C07301=1233.977,-39.079,-38.735,-179.809,5.259,148.853
C07302=1233.971,-38.829,-38.748,-179.806,5.259,148.852
C07303=1233.967,-38.579,-38.761,-179.804,5.260,148.851
C07304=1233.962,-38.330,-38.774,-179.802,5.259,148.851
C07305=1233.956,-38.080,-38.787,-179.799,5.260,148.850
C07306=1233.952,-37.831,-38.800,-179.797,5.260,148.849
C07307=1233.946,-37.581,-38.813,-179.794,5.260,148.849
C07308=1233.941,-37.331,-38.827,-179.792,5.261,148.848
C07309=1233.936,-37.082,-38.839,-179.789,5.260,148.847
C07310=1233.931,-36.832,-38.852,-179.787,5.261,148.846
C07311=1233.926,-36.582,-38.865,-179.785,5.261,148.846
C07312=1233.921,-36.333,-38.879,-179.782,5.261,148.845
C07313=1233.916,-36.083,-38.892,-179.779,5.262,148.844
C07314=1233.910,-35.834,-38.905,-179.777,5.261,148.844
C07315=1233.905,-35.584,-38.917,-179.775,5.262,148.843
C07316=1233.900,-35.334,-38.931,-179.773,5.261,148.842
C07317=1233.895,-35.085,-38.944,-179.769,5.262,148.841
C07318=1233.891,-34.835,-38.957,-179.767,5.262,148.841
C07319=1233.885,-34.586,-38.971,-179.765,5.262,148.840
C07320=1233.880,-34.336,-38.983,-179.762,5.262,148.839
C07321=1233.875,-34.086,-38.997,-179.760,5.262,148.839
C07322=1233.870,-33.837,-39.010,-179.757,5.262,148.838
C07323=1233.865,-33.587,-39.023,-179.755,5.263,148.837
C07324=1233.859,-33.338,-39.036,-179.753,5.263,148.836
C07325=1233.855,-33.088,-39.049,-179.750,5.263,148.836
C07326=1233.849,-32.839,-39.063,-179.748,5.263,148.835
C07327=1233.845,-32.589,-39.076,-179.745,5.263,148.834
C07328=1233.839,-32.339,-39.089,-179.742,5.264,148.834
C07329=1233.835,-32.090,-39.103,-179.740,5.263,148.833
C07330=1233.829,-31.840,-39.116,-179.738,5.264,148.832
C07331=1233.824,-31.590,-39.129,-179.736,5.264,148.832
C07332=1233.819,-31.341,-39.142,-179.733,5.264,148.831
C07333=1233.814,-31.092,-39.156,-179.730,5.265,148.830
C07334=1233.809,-30.842,-39.169,-179.728,5.264,148.829
C07335=1233.803,-30.593,-39.182,-179.725,5.265,148.829
C07336=1233.799,-30.343,-39.195,-179.723,5.264,148.828
C07337=1233.793,-30.093,-39.209,-179.720,5.265,148.827
C07338=1233.789,-29.844,-39.222,-179.718,5.265,148.826
C07339=1233.783,-29.594,-39.235,-179.716,5.265,148.826
C07340=1233.779,-29.344,-39.248,-179.713,5.265,148.825
C07341=1233.773,-29.095,-39.262,-179.711,5.265,148.824
C07342=1233.768,-28.845,-39.275,-179.708,5.266,148.824
C07343=1233.763,-28.596,-39.289,-179.705,5.266,148.823
C07344=1233.758,-28.346,-39.302,-179.703,5.266,148.822
C07345=1233.753,-28.096,-39.316,-179.701,5.266,148.822
C07346=1233.748,-27.846,-39.330,-179.698,5.267,148.821
C07347=1233.743,-27.596,-39.343,-179.696,5.267,148.820
C07348=1233.737,-27.347,-39.357,-179.693,5.267,148.819
C07349=1233.733,-27.097,-39.370,-179.691,5.267,148.819
C07350=1233.727,-26.848,-39.383,-179.689,5.267,148.818
C07351=1233.723,-26.598,-39.396,-179.686,5.268,148.817
C07352=1233.717,-26.349,-39.410,-179.683,5.267,148.816
C07353=1233.713,-26.099,-39.423,-179.681,5.268,148.816
C07354=1233.707,-25.850,-39.437,-179.679,5.267,148.815
C07355=1233.702,-25.600,-39.451,-179.676,5.268,148.814
C07356=1233.698,-25.351,-39.464,-179.673,5.268,148.814
C07357=1233.692,-25.101,-39.478,-179.671,5.268,148.813
C07358=1233.688,-24.852,-39.491,-179.669,5.269,148.812
C07359=1233.682,-24.602,-39.505,-179.666,5.269,148.812
C07360=1233.677,-24.352,-39.519,-179.664,5.269,148.811
C07361=1233.672,-24.103,-39.531,-179.661,5.269,148.810
C07362=1233.667,-23.853,-39.546,-179.659,5.269,148.809
C07363=1233.662,-23.603,-39.559,-179.656,5.269,148.809
C07364=1233.657,-23.354,-39.573,-179.654,5.270,148.808
C07365=1233.652,-23.104,-39.587,-179.652,5.270,148.807
C07366=1233.647,-22.855,-39.599,-179.649,5.270,148.807
C07367=1233.641,-22.586,-39.614,-179.646,5.270,148.806
C07368=1233.636,-22.316,-39.629,-179.643,5.271,148.805
C07369=1233.630,-22.047,-39.644,-179.641,5.271,148.804
C07370=1233.624,-21.778,-39.659,-179.638,5.271,148.804
C07371=1233.620,-21.528,-39.672,-179.635,5.271,148.803
C07372=1233.615,-21.278,-39.686,-179.633,5.271,148.802
C07373=1233.609,-21.029,-39.700,-179.631,5.271,148.801
C07374=1233.605,-20.779,-39.713,-179.628,5.272,148.801
C07375=1233.599,-20.530,-39.727,-179.626,5.272,148.800
C07376=1233.594,-20.281,-39.741,-179.623,5.272,148.799
C07377=1233.590,-20.031,-39.754,-179.620,5.273,148.799
C07378=1233.584,-19.782,-39.768,-179.618,5.272,148.798
C07379=1233.579,-19.532,-39.782,-179.616,5.273,148.797
C07380=1233.574,-19.282,-39.796,-179.614,5.273,148.796
C07381=1233.569,-19.033,-39.809,-179.611,5.273,148.796
C07382=1233.564,-18.783,-39.824,-179.608,5.274,148.795
C07383=1233.559,-18.533,-39.837,-179.606,5.273,148.794
C07384=1233.553,-18.284,-39.851,-179.604,5.274,148.794
C07385=1233.549,-18.035,-39.865,-179.601,5.274,148.793
C07386=1233.544,-17.784,-39.878,-179.599,5.274,148.792
C07387=1233.538,-17.535,-39.892,-179.596,5.275,148.792
C07388=1233.533,-17.285,-39.907,-179.594,5.275,148.791
C07389=1233.529,-17.036,-39.920,-179.591,5.275,148.790
C07390=1233.523,-16.786,-39.933,-179.589,5.275,148.790
C07391=1233.518,-16.537,-39.948,-179.586,5.275,148.789
C07392=1233.513,-16.287,-39.962,-179.584,5.275,148.788
C07393=1233.508,-16.038,-39.976,-179.581,5.276,148.787
C07394=1233.504,-15.789,-39.990,-179.579,5.275,148.787
C07395=1233.498,-15.538,-40.003,-179.576,5.276,148.786
C07396=1233.493,-15.289,-40.017,-179.574,5.276,148.785
C07397=1233.488,-15.040,-40.031,-179.571,5.276,148.784
C07398=1233.483,-14.790,-40.046,-179.569,5.277,148.784
C07399=1233.479,-14.540,-40.059,-179.566,5.277,148.783
C07400=1233.473,-14.291,-40.072,-179.564,5.277,148.782
C07401=1233.468,-14.041,-40.087,-179.561,5.277,148.782
C07402=1233.463,-13.791,-40.101,-179.559,5.278,148.781
C07403=1233.457,-13.542,-40.115,-179.557,5.278,148.780
C07404=1233.452,-13.293,-40.129,-179.554,5.278,148.780
C07405=1233.448,-13.043,-40.143,-179.551,5.279,148.779
C07406=1233.443,-12.794,-40.157,-179.549,5.278,148.778
C07407=1233.438,-12.545,-40.171,-179.547,5.279,148.777
C07408=1233.432,-12.294,-40.185,-179.544,5.279,148.777
C07409=1233.427,-12.045,-40.199,-179.542,5.279,148.776
C07410=1233.422,-11.795,-40.213,-179.539,5.280,148.775
C07411=1233.417,-11.546,-40.227,-179.537,5.280,148.775
C07412=1233.412,-11.296,-40.241,-179.534,5.279,148.774
C07413=1233.408,-11.047,-40.255,-179.531,5.280,148.773
C07414=1233.403,-10.797,-40.269,-179.529,5.280,148.772
C07415=1233.397,-10.548,-40.283,-179.527,5.280,148.772
C07416=1233.392,-10.298,-40.298,-179.524,5.281,148.771
C07417=1233.387,-10.049,-40.312,-179.521,5.281,148.770
C07418=1233.382,-9.799,-40.326,-179.519,5.281,148.770
C07419=1233.377,-9.550,-40.340,-179.517,5.281,148.769
C07420=1233.372,-9.300,-40.354,-179.514,5.282,148.768
C07421=1233.367,-9.050,-40.369,-179.512,5.282,148.768
C07422=1233.362,-8.801,-40.383,-179.509,5.282,148.767
C07423=1233.357,-8.551,-40.397,-179.506,5.283,148.766
C07424=1233.351,-8.302,-40.411,-179.504,5.282,148.765
C07425=1233.346,-8.052,-40.425,-179.502,5.283,148.765
C07426=1233.342,-7.803,-40.440,-179.499,5.283,148.764
C07427=1233.337,-7.553,-40.454,-179.497,5.283,148.763
C07428=1233.332,-7.303,-40.468,-179.494,5.284,148.763
C07429=1233.327,-7.053,-40.482,-179.492,5.284,148.762
C07430=1233.322,-6.805,-40.496,-179.490,5.284,148.761
C07431=1233.317,-6.555,-40.510,-179.487,5.284,148.761
C07432=1233.312,-6.305,-40.524,-179.484,5.285,148.760
C07433=1233.307,-6.056,-40.539,-179.482,5.286,148.759
C07434=1233.302,-5.806,-40.553,-179.480,5.285,148.759
C07435=1233.297,-5.556,-40.567,-179.477,5.286,148.758
C07436=1233.291,-5.307,-40.582,-179.474,5.286,148.757
C07437=1233.286,-5.058,-40.597,-179.472,5.286,148.756
C07438=1233.281,-4.808,-40.611,-179.469,5.286,148.756
C07439=1233.276,-4.558,-40.625,-179.466,5.287,148.755
C07440=1233.271,-4.309,-40.639,-179.464,5.286,148.754
C07441=1233.266,-4.059,-40.654,-179.462,5.287,148.754
C07442=1233.261,-3.810,-40.668,-179.459,5.287,148.753
C07443=1233.256,-3.561,-40.683,-179.457,5.287,148.752
C07444=1233.251,-3.311,-40.697,-179.454,5.288,148.751
C07445=1233.246,-3.061,-40.711,-179.452,5.288,148.751
C07446=1233.241,-2.812,-40.725,-179.450,5.288,148.750
C07447=1233.236,-2.562,-40.740,-179.447,5.288,148.749
C07448=1233.231,-2.312,-40.754,-179.444,5.289,148.749
C07449=1233.227,-2.063,-40.769,-179.442,5.290,148.748
C07450=1233.222,-1.813,-40.783,-179.440,5.289,148.747
C07451=1233.216,-1.564,-40.797,-179.437,5.290,148.747
C07452=1233.210,-1.314,-40.812,-179.434,5.290,148.746
C07453=1233.206,-1.065,-40.827,-179.432,5.290,148.745
C07454=1233.201,-0.816,-40.841,-179.429,5.291,148.745
C07455=1233.196,-0.566,-40.856,-179.427,5.291,148.744
C07456=1233.191,-0.316,-40.870,-179.425,5.291,148.743
C07457=1233.186,-0.067,-40.885,-179.422,5.291,148.742
C07458=1233.181,0.183,-40.899,-179.419,5.292,148.742
C07459=1233.176,0.433,-40.914,-179.417,5.292,148.741
C07460=1233.171,0.682,-40.928,-179.415,5.292,148.740
C07461=1233.166,0.931,-40.943,-179.412,5.293,148.740
C07462=1233.160,1.180,-40.957,-179.409,5.293,148.739
C07463=1233.156,1.430,-40.971,-179.407,5.293,148.738
C07464=1233.151,1.679,-40.986,-179.405,5.293,148.738
C07465=1233.145,1.929,-41.001,-179.402,5.294,148.737
C07466=1233.140,2.179,-41.016,-179.399,5.294,148.736
C07467=1233.136,2.428,-41.031,-179.397,5.294,148.736
C07468=1233.131,2.678,-41.045,-179.395,5.295,148.735
C07469=1233.126,2.927,-41.059,-179.392,5.295,148.734
C07470=1233.120,3.177,-41.075,-179.389,5.295,148.733
C07471=1233.115,3.446,-41.090,-179.387,5.295,148.733
C07472=1233.110,3.714,-41.106,-179.384,5.296,148.732
C07473=1233.105,3.983,-41.122,-179.381,5.296,148.731
C07474=1233.099,4.252,-41.138,-179.378,5.296,148.730
C07475=1233.094,4.502,-41.152,-179.376,5.297,148.730
C07476=1233.089,4.752,-41.167,-179.374,5.297,148.729
C07477=1233.084,5.001,-41.182,-179.371,5.297,148.728
C07478=1233.079,5.251,-41.197,-179.368,5.298,148.728
C07479=1233.074,5.500,-41.212,-179.366,5.297,148.727
C07480=1233.069,5.750,-41.226,-179.364,5.298,148.726
C07481=1233.065,5.999,-41.241,-179.361,5.299,148.725
C07482=1233.059,6.249,-41.256,-179.358,5.299,148.725
C07483=1233.054,6.498,-41.271,-179.356,5.299,148.724
C07484=1233.049,6.748,-41.285,-179.354,5.299,148.723
C07485=1233.044,6.998,-41.300,-179.351,5.300,148.723
C07486=1233.039,7.247,-41.315,-179.349,5.300,148.722
C07487=1233.034,7.496,-41.329,-179.346,5.300,148.721
C07488=1233.029,7.746,-41.344,-179.343,5.301,148.721
C07489=1233.024,7.995,-41.360,-179.341,5.301,148.720
C07490=1233.019,8.245,-41.374,-179.339,5.301,148.719
C07491=1233.014,8.494,-41.389,-179.336,5.301,148.719
C07492=1233.009,8.744,-41.404,-179.333,5.302,148.718
C07493=1233.004,8.993,-41.419,-179.331,5.303,148.717
C07494=1232.999,9.243,-41.433,-179.329,5.302,148.717
C07495=1232.994,9.492,-41.449,-179.326,5.303,148.716
C07496=1232.989,9.742,-41.463,-179.323,5.303,148.715
C07497=1232.984,9.991,-41.478,-179.321,5.304,148.715
C07498=1232.979,10.240,-41.494,-179.319,5.304,148.714
C07499=1232.974,10.490,-41.508,-179.316,5.304,148.713
C07500=1232.968,10.739,-41.523,-179.313,5.305,148.712
C07501=1232.964,10.990,-41.538,-179.311,5.305,148.712
C07502=1232.959,11.239,-41.553,-179.309,5.305,148.711
C07503=1232.954,11.488,-41.569,-179.306,5.305,148.710
C07504=1232.949,11.738,-41.583,-179.303,5.306,148.710
C07505=1232.944,11.987,-41.599,-179.301,5.306,148.709
C07506=1232.939,12.236,-41.614,-179.299,5.306,148.708
C07507=1232.934,12.486,-41.628,-179.296,5.307,148.708
C07508=1232.929,12.735,-41.643,-179.293,5.307,148.707
C07509=1232.924,12.985,-41.658,-179.291,5.307,148.706
C07510=1232.918,13.235,-41.673,-179.289,5.308,148.706
C07511=1232.914,13.484,-41.688,-179.286,5.308,148.705
C07512=1232.910,13.733,-41.704,-179.283,5.309,148.704
C07513=1232.904,13.983,-41.718,-179.281,5.308,148.704
C07514=1232.899,14.233,-41.733,-179.279,5.309,148.703
C07515=1232.894,14.482,-41.749,-179.276,5.310,148.702
C07516=1232.889,14.732,-41.763,-179.273,5.310,148.701
C07517=1232.883,14.981,-41.779,-179.271,5.310,148.701
C07518=1232.879,15.230,-41.794,-179.269,5.310,148.700
C07519=1232.874,15.480,-41.810,-179.266,5.311,148.699
C07520=1232.869,15.730,-41.824,-179.263,5.311,148.699
C07521=1232.864,15.979,-41.840,-179.261,5.312,148.698
C07522=1232.859,16.228,-41.855,-179.259,5.312,148.697
C07523=1232.854,16.478,-41.870,-179.256,5.312,148.697
C07524=1232.849,16.727,-41.885,-179.253,5.313,148.696
C07525=1232.843,16.977,-41.900,-179.251,5.313,148.695
C07526=1232.839,17.227,-41.916,-179.249,5.313,148.695
C07527=1232.834,17.476,-41.931,-179.246,5.314,148.694
C07528=1232.829,17.725,-41.946,-179.243,5.314,148.693
C07529=1232.824,17.975,-41.962,-179.241,5.315,148.693
C07530=1232.819,18.224,-41.976,-179.239,5.314,148.692
C07531=1232.814,18.474,-41.992,-179.236,5.315,148.691
C07532=1232.809,18.724,-42.007,-179.233,5.316,148.691
C07533=1232.804,18.973,-42.023,-179.231,5.316,148.690
C07534=1232.799,19.222,-42.038,-179.228,5.317,148.689
C07535=1232.794,19.472,-42.053,-179.226,5.316,148.688
C07536=1232.789,19.721,-42.069,-179.223,5.317,148.688
C07537=1232.785,19.971,-42.084,-179.221,5.317,148.687
C07538=1232.779,20.221,-42.099,-179.218,5.318,148.686
C07539=1232.774,20.470,-42.114,-179.216,5.318,148.686
C07540=1232.769,20.719,-42.130,-179.213,5.318,148.685
C07541=1232.763,20.969,-42.145,-179.211,5.319,148.684
C07542=1232.759,21.218,-42.160,-179.208,5.319,148.684
C07543=1232.754,21.468,-42.176,-179.205,5.320,148.683
C07544=1232.749,21.717,-42.191,-179.203,5.320,148.682
C07545=1232.744,21.966,-42.207,-179.201,5.320,148.682
C07546=1232.739,22.216,-42.223,-179.198,5.321,148.681
C07547=1232.735,22.465,-42.238,-179.195,5.321,148.680
C07548=1232.729,22.715,-42.253,-179.193,5.321,148.680
C07549=1232.724,22.964,-42.269,-179.191,5.322,148.679
C07550=1232.720,23.214,-42.284,-179.188,5.322,148.678
C07551=1232.714,23.464,-42.300,-179.185,5.323,148.678
C07552=1232.709,23.713,-42.315,-179.183,5.323,148.677
C07553=1232.704,23.962,-42.330,-179.181,5.323,148.676
C07554=1232.700,24.212,-42.346,-179.178,5.324,148.676
C07555=1232.694,24.462,-42.362,-179.175,5.324,148.675
C07556=1232.690,24.711,-42.377,-179.173,5.325,148.674
C07557=1232.684,24.960,-42.392,-179.170,5.325,148.674
C07558=1232.679,25.210,-42.408,-179.168,5.325,148.673
C07559=1232.675,25.459,-42.423,-179.165,5.325,148.672
C07560=1232.669,25.709,-42.439,-179.163,5.326,148.671
C07561=1232.665,25.959,-42.455,-179.160,5.327,148.671
C07562=1232.660,26.207,-42.471,-179.158,5.327,148.670
C07563=1232.655,26.457,-42.486,-179.156,5.327,148.670
C07564=1232.650,26.707,-42.502,-179.153,5.328,148.669
C07565=1232.645,26.956,-42.518,-179.150,5.328,148.668
C07566=1232.640,27.205,-42.533,-179.148,5.329,148.668
C07567=1232.635,27.455,-42.548,-179.145,5.329,148.667
C07568=1232.630,27.705,-42.564,-179.143,5.329,148.666
C07569=1232.624,27.954,-42.580,-179.140,5.330,148.666
C07570=1232.620,28.203,-42.596,-179.138,5.330,148.665
C07571=1232.615,28.453,-42.612,-179.135,5.331,148.664
C07572=1232.610,28.702,-42.627,-179.132,5.331,148.664
C07573=1232.605,28.951,-42.643,-179.130,5.331,148.663
C07574=1232.600,29.202,-42.659,-179.128,5.332,148.662
C07575=1232.595,29.470,-42.675,-179.125,5.332,148.661
C07576=1232.589,29.738,-42.692,-179.122,5.332,148.661
C07577=1232.584,30.007,-42.709,-179.119,5.333,148.660
C07578=1232.578,30.275,-42.726,-179.117,5.334,148.659
C07579=1232.573,30.525,-42.742,-179.114,5.334,148.659
C07580=1232.568,30.775,-42.758,-179.111,5.335,148.658
C07581=1232.564,31.024,-42.774,-179.109,5.334,148.657
C07582=1232.559,31.273,-42.789,-179.107,5.335,148.657
C07583=1232.554,31.523,-42.805,-179.104,5.336,148.656
C07584=1232.549,31.772,-42.822,-179.101,5.336,148.655
C07585=1232.544,32.022,-42.837,-179.099,5.337,148.654
C07586=1232.538,32.271,-42.853,-179.096,5.337,148.654
C07587=1232.534,32.521,-42.868,-179.094,5.337,148.653
C07588=1232.529,32.770,-42.884,-179.091,5.337,148.652
C07589=1232.524,33.020,-42.900,-179.089,5.338,148.652
C07590=1232.519,33.269,-42.916,-179.087,5.339,148.651
C07591=1232.514,33.518,-42.932,-179.084,5.340,148.651
C07592=1232.509,33.768,-42.948,-179.081,5.340,148.650
C07593=1232.504,34.017,-42.964,-179.079,5.340,148.649
C07594=1232.499,34.267,-42.980,-179.077,5.340,148.649
C07595=1232.494,34.516,-42.996,-179.074,5.341,148.648
C07596=1232.489,34.765,-43.011,-179.071,5.341,148.647
C07597=1232.485,35.015,-43.028,-179.069,5.342,148.647
C07598=1232.479,35.264,-43.043,-179.066,5.343,148.646
C07599=1232.475,35.514,-43.060,-179.064,5.342,148.645
C07600=1232.469,35.763,-43.076,-179.061,5.343,148.645
C07601=1232.465,36.013,-43.092,-179.059,5.343,148.644
C07602=1232.460,36.262,-43.108,-179.056,5.344,148.643
C07603=1232.455,36.512,-43.124,-179.053,5.345,148.643
C07604=1232.450,36.761,-43.140,-179.051,5.345,148.642
C07605=1232.444,37.010,-43.156,-179.049,5.345,148.641
C07606=1232.440,37.260,-43.172,-179.046,5.345,148.640
C07607=1232.434,37.509,-43.188,-179.043,5.346,148.640
C07608=1232.430,37.759,-43.204,-179.041,5.347,148.639
C07609=1232.425,38.008,-43.220,-179.039,5.348,148.639
C07610=1232.420,38.258,-43.236,-179.036,5.348,148.638
C07611=1232.415,38.507,-43.252,-179.034,5.348,148.637
C07612=1232.410,38.757,-43.268,-179.031,5.348,148.637
C07613=1232.405,39.006,-43.285,-179.029,5.349,148.636
C07614=1232.400,39.256,-43.301,-179.026,5.350,148.635
C07615=1232.395,39.505,-43.317,-179.023,5.350,148.635
C07616=1232.390,39.755,-43.333,-179.021,5.351,148.634
C07617=1232.385,40.004,-43.349,-179.018,5.351,148.633
C07618=1232.380,40.254,-43.365,-179.016,5.351,148.633
C07619=1232.375,40.502,-43.381,-179.013,5.352,148.632
C07620=1232.371,40.752,-43.398,-179.011,5.352,148.631
C07621=1232.365,41.001,-43.414,-179.008,5.353,148.631
C07622=1232.361,41.251,-43.430,-179.005,5.353,148.630
C07623=1232.356,41.500,-43.446,-179.003,5.354,148.629
C07624=1232.351,41.750,-43.463,-179.001,5.355,148.629
C07625=1232.346,41.998,-43.479,-178.998,5.355,148.628
C07626=1232.341,42.249,-43.495,-178.996,5.355,148.627
C07627=1232.335,42.498,-43.512,-178.993,5.356,148.627
C07628=1232.331,42.748,-43.528,-178.991,5.356,148.626
C07629=1232.326,42.997,-43.544,-178.988,5.357,148.625
C07630=1232.321,43.246,-43.561,-178.985,5.357,148.625
C07631=1232.316,43.495,-43.576,-178.983,5.358,148.624
C07632=1232.311,43.745,-43.593,-178.980,5.358,148.623
C07633=1232.307,43.994,-43.610,-178.978,5.358,148.623
C07634=1232.301,44.244,-43.625,-178.975,5.359,148.622
C07635=1232.297,44.493,-43.642,-178.973,5.359,148.621
C07636=1232.291,44.742,-43.659,-178.970,5.360,148.621
C07637=1232.286,44.993,-43.675,-178.967,5.360,148.620
C07638=1232.281,45.241,-43.691,-178.965,5.361,148.620
C07639=1232.277,45.491,-43.708,-178.963,5.362,148.619
C07640=1232.272,45.740,-43.724,-178.960,5.363,148.618
C07641=1232.267,45.990,-43.740,-178.958,5.362,148.618
C07642=1232.262,46.239,-43.757,-178.955,5.363,148.617
C07643=1232.256,46.488,-43.774,-178.953,5.363,148.616
C07644=1232.252,46.738,-43.790,-178.950,5.364,148.616
C07645=1232.247,46.988,-43.806,-178.947,5.365,148.615
C07646=1232.242,47.237,-43.822,-178.945,5.365,148.614
C07647=1232.238,47.486,-43.839,-178.942,5.366,148.614
C07648=1232.232,47.735,-43.856,-178.940,5.366,148.613
C07649=1232.227,47.985,-43.872,-178.937,5.367,148.612
C07650=1232.223,48.235,-43.889,-178.935,5.367,148.612
C07651=1232.218,48.484,-43.905,-178.933,5.368,148.611
C07652=1232.212,48.733,-43.922,-178.930,5.368,148.610
C07653=1232.207,48.982,-43.939,-178.927,5.369,148.610
C07654=1232.203,49.232,-43.955,-178.925,5.369,148.609
C07655=1232.198,49.482,-43.971,-178.922,5.370,148.608
C07656=1232.192,49.731,-43.988,-178.919,5.370,148.608
C07657=1232.188,49.980,-44.005,-178.917,5.371,148.607
C07658=1232.183,50.230,-44.021,-178.914,5.372,148.606
C07659=1232.178,50.479,-44.038,-178.912,5.372,148.606
C07660=1232.173,50.728,-44.055,-178.910,5.372,148.605
C07661=1232.168,50.978,-44.072,-178.907,5.373,148.605
C07662=1232.163,51.227,-44.088,-178.905,5.373,148.604
C07663=1232.159,51.477,-44.104,-178.902,5.374,148.603
C07664=1232.153,51.727,-44.121,-178.899,5.375,148.603
C07665=1232.148,51.975,-44.137,-178.897,5.375,148.602
C07666=1232.144,52.225,-44.154,-178.894,5.376,148.601
C07667=1232.139,52.475,-44.171,-178.892,5.376,148.601
C07668=1232.133,52.723,-44.188,-178.889,5.377,148.600
C07669=1232.129,52.973,-44.204,-178.886,5.377,148.599
C07670=1232.124,53.223,-44.222,-178.884,5.378,148.599
C07671=1232.119,53.472,-44.238,-178.882,5.378,148.598
C07672=1232.114,53.721,-44.255,-178.879,5.379,148.597
C07673=1232.109,53.971,-44.272,-178.877,5.379,148.597
C07674=1232.104,54.220,-44.289,-178.874,5.380,148.596
C07675=1232.099,54.469,-44.305,-178.872,5.380,148.595
C07676=1232.094,54.719,-44.322,-178.869,5.381,148.595
C07677=1232.090,54.968,-44.339,-178.866,5.382,148.594
C07678=1232.085,55.217,-44.355,-178.864,5.382,148.593
C07679=1232.079,55.486,-44.374,-178.861,5.383,148.593
C07680=1232.075,55.754,-44.392,-178.858,5.383,148.592
C07681=1232.069,56.023,-44.410,-178.856,5.384,148.591
C07682=1232.064,56.291,-44.428,-178.853,5.384,148.591
C07683=1232.058,56.540,-44.445,-178.850,5.385,148.590
C07684=1232.054,56.790,-44.462,-178.848,5.386,148.589
C07685=1232.048,57.040,-44.479,-178.845,5.386,148.589
C07686=1232.044,57.289,-44.496,-178.843,5.387,148.588
C07687=1232.039,57.538,-44.512,-178.840,5.388,148.588
C07688=1232.034,57.788,-44.529,-178.838,5.388,148.587
C07689=1232.029,58.037,-44.547,-178.835,5.389,148.586
C07690=1232.024,58.286,-44.564,-178.833,5.389,148.586
C07691=1232.019,58.535,-44.580,-178.830,5.390,148.585
C07692=1232.014,58.785,-44.598,-178.828,5.390,148.584
C07693=1232.009,59.034,-44.614,-178.825,5.390,148.584
C07694=1232.004,59.284,-44.632,-178.823,5.391,148.583
C07695=1232.000,59.533,-44.649,-178.820,5.392,148.583
C07696=1231.994,59.782,-44.666,-178.818,5.392,148.582
C07697=1231.990,60.032,-44.682,-178.815,5.393,148.581
C07698=1231.985,60.281,-44.700,-178.813,5.394,148.581
C07699=1231.980,60.531,-44.716,-178.810,5.394,148.580
C07700=1231.975,60.780,-44.734,-178.807,5.395,148.579
C07701=1231.970,61.029,-44.751,-178.805,5.395,148.579
C07702=1231.965,61.279,-44.768,-178.802,5.396,148.578
C07703=1231.960,61.528,-44.785,-178.800,5.397,148.578
C07704=1231.955,61.777,-44.803,-178.797,5.397,148.577
C07705=1231.951,62.027,-44.819,-178.795,5.398,148.576
C07706=1231.945,62.276,-44.836,-178.792,5.399,148.576
C07707=1231.941,62.525,-44.853,-178.789,5.399,148.575
C07708=1231.936,62.775,-44.871,-178.787,5.400,148.574
C07709=1231.931,63.024,-44.888,-178.785,5.401,148.574
C07710=1231.926,63.274,-44.905,-178.782,5.401,148.573
C07711=1231.921,63.523,-44.923,-178.779,5.402,148.572
C07712=1231.917,63.772,-44.939,-178.777,5.402,148.572
C07713=1231.911,64.022,-44.956,-178.775,5.402,148.571
C07714=1231.907,64.270,-44.974,-178.772,5.403,148.570
C07715=1231.901,64.520,-44.991,-178.769,5.403,148.570
C07716=1231.896,64.770,-45.008,-178.767,5.404,148.569
C07717=1231.892,65.019,-45.026,-178.765,5.405,148.569
C07718=1231.887,65.269,-45.043,-178.762,5.406,148.568
C07719=1231.882,65.518,-45.060,-178.759,5.406,148.567
C07720=1231.877,65.767,-45.078,-178.757,5.407,148.567
C07721=1231.872,66.016,-45.094,-178.754,5.407,148.566
C07722=1231.867,66.265,-45.112,-178.751,5.408,148.565
C07723=1231.862,66.515,-45.129,-178.749,5.409,148.565
C07724=1231.857,66.764,-45.147,-178.747,5.409,148.564
C07725=1231.853,67.014,-45.164,-178.744,5.410,148.564
C07726=1231.848,67.264,-45.181,-178.741,5.411,148.563
C07727=1231.843,67.513,-45.199,-178.739,5.411,148.562
C07728=1231.838,67.762,-45.216,-178.736,5.412,148.562
C07729=1231.833,68.011,-45.234,-178.734,5.413,148.561
C07730=1231.828,68.261,-45.251,-178.731,5.413,148.560
C07731=1231.824,68.510,-45.268,-178.729,5.414,148.560
C07732=1231.818,68.759,-45.285,-178.726,5.414,148.559
C07733=1231.813,69.008,-45.303,-178.723,5.415,148.559
C07734=1231.809,69.258,-45.320,-178.721,5.416,148.558
C07735=1231.804,69.507,-45.338,-178.719,5.417,148.557
C07736=1231.799,69.757,-45.355,-178.716,5.417,148.557
C07737=1231.794,70.006,-45.373,-178.713,5.418,148.556
C07738=1231.789,70.255,-45.390,-178.711,5.418,148.555
C07739=1231.784,70.505,-45.408,-178.708,5.419,148.555
C07740=1231.779,70.754,-45.426,-178.706,5.420,148.554
C07741=1231.775,71.003,-45.442,-178.703,5.420,148.554
C07742=1231.770,71.252,-45.460,-178.701,5.421,148.553
C07743=1231.765,71.502,-45.478,-178.698,5.422,148.552
C07744=1231.760,71.751,-45.496,-178.696,5.422,148.552
C07745=1231.755,72.001,-45.513,-178.693,5.423,148.551
C07746=1231.751,72.250,-45.530,-178.690,5.423,148.550
C07747=1231.746,72.499,-45.548,-178.688,5.424,148.550
C07748=1231.740,72.749,-45.565,-178.685,5.425,148.549
C07749=1231.735,72.998,-45.583,-178.683,5.426,148.549
C07750=1231.731,73.247,-45.601,-178.680,5.426,148.548
C07751=1231.726,73.497,-45.618,-178.678,5.427,148.547
C07752=1231.721,73.746,-45.636,-178.675,5.428,148.547
C07753=1231.716,73.995,-45.654,-178.673,5.428,148.546
C07754=1231.711,74.245,-45.671,-178.670,5.429,148.546
C07755=1231.706,74.494,-45.689,-178.668,5.429,148.545
C07756=1231.702,74.743,-45.707,-178.665,5.430,148.544
C07757=1231.697,74.993,-45.724,-178.662,5.431,148.544
C07758=1231.692,75.242,-45.742,-178.660,5.432,148.543
C07759=1231.687,75.491,-45.760,-178.658,5.432,148.542
C07760=1231.682,75.740,-45.778,-178.655,5.433,148.542
C07761=1231.677,75.990,-45.795,-178.652,5.433,148.541
C07762=1231.672,76.239,-45.813,-178.650,5.434,148.541
C07763=1231.667,76.489,-45.831,-178.648,5.435,148.540
C07764=1231.663,76.737,-45.848,-178.645,5.436,148.539
C07765=1231.658,76.987,-45.866,-178.642,5.436,148.539
C07766=1231.653,77.236,-45.884,-178.640,5.437,148.538
C07767=1231.648,77.486,-45.902,-178.637,5.437,148.537
C07768=1231.643,77.735,-45.920,-178.635,5.438,148.537
C07769=1231.639,77.985,-45.938,-178.632,5.439,148.536
C07770=1231.633,78.234,-45.955,-178.630,5.439,148.536
C07771=1231.628,78.484,-45.973,-178.627,5.440,148.535
C07772=1231.623,78.733,-45.991,-178.624,5.441,148.534
C07773=1231.619,78.982,-46.009,-178.622,5.442,148.534
C07774=1231.614,79.231,-46.027,-178.620,5.442,148.533
C07775=1231.609,79.480,-46.045,-178.617,5.443,148.533
C07776=1231.604,79.730,-46.062,-178.614,5.443,148.532
C07777=1231.599,79.979,-46.080,-178.612,5.444,148.531
C07778=1231.594,80.228,-46.098,-178.609,5.446,148.531
C07779=1231.590,80.477,-46.116,-178.606,5.446,148.530
C07780=1231.585,80.727,-46.134,-178.604,5.447,148.530
C07781=1231.580,80.976,-46.152,-178.601,5.448,148.529
C07782=1231.575,81.226,-46.170,-178.599,5.448,148.529
C07783=1231.570,81.494,-46.190,-178.596,5.449,148.528
C07784=1231.564,81.762,-46.210,-178.594,5.450,148.527
C07785=1231.559,82.031,-46.228,-178.591,5.450,148.527
C07786=1231.554,82.299,-46.248,-178.589,5.451,148.526
C07787=1231.549,82.549,-46.266,-178.585,5.452,148.525
C07788=1231.544,82.798,-46.284,-178.583,5.453,148.525
C07789=1231.539,83.047,-46.302,-178.580,5.454,148.524
C07790=1231.534,83.296,-46.320,-178.578,5.454,148.523
C07791=1231.529,83.545,-46.338,-178.575,5.455,148.523
C07792=1231.525,83.795,-46.356,-178.573,5.456,148.522
C07793=1231.520,84.044,-46.374,-178.570,5.456,148.522
C07794=1231.515,84.294,-46.392,-178.568,5.457,148.521
C07795=1231.510,84.543,-46.410,-178.565,5.458,148.520
C07796=1231.505,84.792,-46.428,-178.563,5.458,148.520
C07797=1231.500,85.041,-46.446,-178.560,5.459,148.519
C07798=1231.496,85.291,-46.465,-178.558,5.460,148.519
C07799=1231.491,85.540,-46.483,-178.555,5.461,148.518
C07800=1231.486,85.789,-46.501,-178.553,5.461,148.517
C07801=1231.481,86.038,-46.519,-178.550,5.462,148.517
C07802=1231.476,86.287,-46.537,-178.548,5.462,148.516
C07803=1231.472,86.537,-46.556,-178.544,5.464,148.515
C07804=1231.467,86.786,-46.574,-178.542,5.465,148.515
C07805=1231.462,87.036,-46.592,-178.540,5.465,148.514
C07806=1231.456,87.285,-46.610,-178.537,5.466,148.514
C07807=1231.452,87.535,-46.629,-178.534,5.467,148.513
C07808=1231.447,87.784,-46.647,-178.532,5.468,148.513
C07809=1231.443,88.033,-46.665,-178.530,5.468,148.512
C07810=1231.438,88.282,-46.683,-178.527,5.469,148.511
C07811=1231.433,88.531,-46.701,-178.524,5.469,148.511
C07812=1231.428,88.781,-46.720,-178.522,5.470,148.510
C07813=1231.423,89.030,-46.738,-178.520,5.471,148.510
C07814=1231.418,89.279,-46.757,-178.517,5.472,148.509
C07815=1231.413,89.528,-46.775,-178.514,5.472,148.508
C07816=1231.409,89.778,-46.793,-178.512,5.474,148.508
C07817=1231.403,90.027,-46.812,-178.509,5.475,148.507
C07818=1231.399,90.276,-46.830,-178.506,5.475,148.507
C07819=1231.394,90.525,-46.848,-178.504,5.476,148.506
C07820=1231.389,90.775,-46.867,-178.502,5.477,148.506
C07821=1231.385,91.024,-46.885,-178.499,5.477,148.505
C07822=1231.379,91.273,-46.904,-178.496,5.478,148.504
C07823=1231.375,91.523,-46.922,-178.494,5.479,148.504
C07824=1231.370,91.772,-46.940,-178.492,5.479,148.503
C07825=1231.365,92.021,-46.958,-178.489,5.480,148.502
C07826=1231.360,92.270,-46.978,-178.486,5.482,148.502
C07827=1231.355,92.520,-46.996,-178.484,5.482,148.501
C07828=1231.351,92.769,-47.014,-178.481,5.483,148.501
C07829=1231.346,93.018,-47.033,-178.478,5.484,148.500
C07830=1231.341,93.268,-47.052,-178.476,5.484,148.499
C07831=1231.336,93.517,-47.070,-178.474,5.485,148.499
C07832=1231.331,93.766,-47.088,-178.471,5.486,148.498
C07833=1231.326,94.016,-47.107,-178.468,5.486,148.498
C07834=1231.322,94.265,-47.126,-178.466,5.487,148.497
C07835=1231.317,94.514,-47.144,-178.463,5.489,148.497
C07836=1231.312,94.764,-47.163,-178.461,5.489,148.496
C07837=1231.307,95.012,-47.181,-178.458,5.490,148.495
C07838=1231.302,95.262,-47.199,-178.456,5.491,148.495
C07839=1231.297,95.511,-47.219,-178.453,5.492,148.494
C07840=1231.293,95.760,-47.237,-178.451,5.492,148.494
C07841=1231.288,96.010,-47.255,-178.448,5.493,148.493
C07842=1231.283,96.259,-47.275,-178.446,5.494,148.493
C07843=1231.278,96.508,-47.293,-178.443,5.494,148.492
C07844=1231.273,96.757,-47.311,-178.440,5.496,148.491
C07845=1231.268,97.007,-47.330,-178.437,5.496,148.491
C07846=1231.264,97.256,-47.349,-178.435,5.497,148.490
C07847=1231.258,97.505,-47.368,-178.433,5.498,148.490
C07848=1231.254,97.754,-47.387,-178.430,5.499,148.489
C07849=1231.249,98.003,-47.405,-178.428,5.500,148.489
C07850=1231.244,98.253,-47.424,-178.425,5.500,148.488
C07851=1231.240,98.502,-47.442,-178.423,5.501,148.487
C07852=1231.234,98.751,-47.462,-178.420,5.503,148.487
C07853=1231.230,99.001,-47.480,-178.417,5.503,148.486
C07854=1231.225,99.250,-47.499,-178.415,5.504,148.486
C07855=1231.221,99.499,-47.518,-178.412,5.504,148.485
C07856=1231.216,99.748,-47.536,-178.410,5.505,148.484
C07857=1231.210,99.997,-47.556,-178.407,5.506,148.484
C07858=1231.206,100.247,-47.574,-178.405,5.507,148.483
C07859=1231.201,100.496,-47.593,-178.402,5.508,148.483
C07860=1231.196,100.746,-47.612,-178.399,5.509,148.482
C07861=1231.191,100.995,-47.631,-178.397,5.510,148.481
C07862=1231.186,101.243,-47.650,-178.395,5.511,148.481
C07863=1231.181,101.493,-47.668,-178.392,5.511,148.480
C07864=1231.177,101.742,-47.687,-178.390,5.512,148.480
C07865=1231.172,101.992,-47.707,-178.387,5.513,148.479
C07866=1231.167,102.241,-47.725,-178.384,5.514,148.479
C07867=1231.162,102.490,-47.744,-178.382,5.515,148.478
C07868=1231.158,102.739,-47.763,-178.379,5.516,148.477
C07869=1231.153,102.989,-47.782,-178.377,5.516,148.477
C07870=1231.148,103.238,-47.801,-178.374,5.517,148.476
C07871=1231.143,103.487,-47.820,-178.372,5.518,148.476
C07872=1231.138,103.736,-47.838,-178.369,5.520,148.475
C07873=1231.133,103.985,-47.858,-178.366,5.520,148.475
C07874=1231.129,104.234,-47.877,-178.364,5.521,148.474
C07875=1231.124,104.483,-47.896,-178.362,5.522,148.474
C07876=1231.119,104.733,-47.915,-178.359,5.522,148.473
C07877=1231.114,104.982,-47.934,-178.356,5.523,148.472
C07878=1231.109,105.232,-47.953,-178.354,5.525,148.472
C07879=1231.105,105.480,-47.972,-178.351,5.525,148.471
C07880=1231.100,105.730,-47.992,-178.348,5.526,148.471
C07881=1231.095,105.979,-48.010,-178.346,5.527,148.470
C07882=1231.090,106.228,-48.029,-178.344,5.528,148.470
C07883=1231.085,106.477,-48.049,-178.341,5.528,148.469
C07884=1231.081,106.727,-48.068,-178.338,5.530,148.469
C07885=1231.076,106.975,-48.087,-178.336,5.531,148.468
C07886=1231.071,107.226,-48.106,-178.333,5.531,148.467
C07887=1231.066,107.494,-48.126,-178.331,5.532,148.467
C07888=1231.061,107.762,-48.147,-178.328,5.534,148.466
C07889=1231.056,108.031,-48.168,-178.325,5.534,148.466
C07890=1231.050,108.299,-48.188,-178.323,5.535,148.465
C07891=1231.045,108.549,-48.208,-178.319,5.536,148.464
C07892=1231.041,108.797,-48.227,-178.317,5.537,148.464
C07893=1231.036,109.047,-48.246,-178.315,5.538,148.463
C07894=1231.031,109.296,-48.266,-178.312,5.539,148.463
C07895=1231.027,109.545,-48.285,-178.310,5.540,148.462
C07896=1231.022,109.795,-48.304,-178.307,5.541,148.462
C07897=1231.017,110.043,-48.324,-178.304,5.542,148.461
C07898=1231.012,110.293,-48.343,-178.302,5.543,148.460
C07899=1231.007,110.542,-48.362,-178.299,5.543,148.460
C07900=1231.002,110.791,-48.382,-178.297,5.544,148.459
C07901=1230.997,111.040,-48.401,-178.294,5.546,148.459
C07902=1230.993,111.289,-48.420,-178.292,5.546,148.458
C07903=1230.988,111.539,-48.440,-178.289,5.547,148.457
C07904=1230.983,111.788,-48.459,-178.287,5.548,148.457
C07905=1230.978,112.037,-48.479,-178.284,5.548,148.456
C07906=1230.974,112.286,-48.497,-178.281,5.550,148.456
C07907=1230.969,112.535,-48.517,-178.279,5.551,148.455
C07908=1230.964,112.785,-48.537,-178.276,5.551,148.455
C07909=1230.959,113.034,-48.556,-178.274,5.552,148.454
C07910=1230.955,113.283,-48.575,-178.272,5.553,148.454
C07911=1230.950,113.533,-48.595,-178.268,5.555,148.453
C07912=1230.945,113.781,-48.614,-178.266,5.555,148.453
C07913=1230.940,114.031,-48.633,-178.264,5.556,148.452
C07914=1230.935,114.280,-48.653,-178.261,5.557,148.451
C07915=1230.930,114.529,-48.672,-178.259,5.558,148.451
C07916=1230.926,114.779,-48.691,-178.256,5.559,148.450
C07917=1230.921,115.027,-48.711,-178.253,5.560,148.450
C07918=1230.916,115.277,-48.731,-178.251,5.561,148.449
C07919=1230.911,115.526,-48.751,-178.248,5.561,148.449
C07920=1230.906,115.775,-48.770,-178.246,5.563,148.448
C07921=1230.901,116.025,-48.790,-178.243,5.564,148.448
C07922=1230.897,116.274,-48.809,-178.241,5.564,148.447
C07923=1230.892,116.523,-48.828,-178.238,5.565,148.447
C07924=1230.888,116.772,-48.848,-178.236,5.566,148.446
C07925=1230.883,117.021,-48.868,-178.233,5.568,148.446
C07926=1230.877,117.270,-48.887,-178.231,5.568,148.445
C07927=1230.873,117.520,-48.907,-178.228,5.569,148.444
C07928=1230.868,117.769,-48.927,-178.226,5.570,148.444
C07929=1230.863,118.017,-48.947,-178.223,5.572,148.443
C07930=1230.858,118.267,-48.966,-178.220,5.572,148.443
C07931=1230.854,118.516,-48.985,-178.218,5.573,148.442
C07932=1230.849,118.766,-49.005,-178.215,5.574,148.442
C07933=1230.844,119.014,-49.025,-178.213,5.576,148.441
C07934=1230.840,119.264,-49.045,-178.210,5.576,148.441
C07935=1230.835,119.513,-49.064,-178.207,5.577,148.440
C07936=1230.830,119.761,-49.084,-178.205,5.578,148.439
C07937=1230.825,120.011,-49.104,-178.202,5.579,148.439
C07938=1230.820,120.261,-49.124,-178.200,5.580,148.438
C07939=1230.816,120.510,-49.144,-178.197,5.581,148.438
C07940=1230.811,120.758,-49.163,-178.195,5.581,148.437
C07941=1230.806,121.008,-49.183,-178.192,5.583,148.437
C07942=1230.801,121.257,-49.203,-178.189,5.584,148.436
C07943=1230.797,121.507,-49.223,-178.187,5.585,148.436
C07944=1230.791,121.755,-49.242,-178.185,5.586,148.435
C07945=1230.787,122.004,-49.263,-178.182,5.587,148.435
C07946=1230.782,122.254,-49.282,-178.179,5.588,148.434
C07947=1230.777,122.503,-49.302,-178.177,5.589,148.433
C07948=1230.772,122.752,-49.322,-178.175,5.590,148.433
C07949=1230.768,123.001,-49.342,-178.172,5.591,148.432
C07950=1230.763,123.250,-49.362,-178.169,5.592,148.432
C07951=1230.758,123.500,-49.382,-178.167,5.593,148.431
C07952=1230.754,123.749,-49.402,-178.164,5.594,148.431
C07953=1230.749,123.998,-49.421,-178.162,5.595,148.430
C07954=1230.744,124.247,-49.442,-178.159,5.596,148.430
C07955=1230.739,124.496,-49.461,-178.157,5.597,148.429
C07956=1230.735,124.746,-49.481,-178.154,5.598,148.429
C07957=1230.730,124.995,-49.501,-178.152,5.599,148.428
C07958=1230.725,125.244,-49.521,-178.149,5.600,148.428
C07959=1230.720,125.493,-49.542,-178.146,5.600,148.427
C07960=1230.715,125.742,-49.561,-178.144,5.602,148.427
C07961=1230.711,125.991,-49.582,-178.141,5.603,148.426
C07962=1230.706,126.240,-49.602,-178.139,5.604,148.426
C07963=1230.701,126.490,-49.622,-178.136,5.605,148.425
C07964=1230.696,126.738,-49.642,-178.134,5.606,148.425
C07965=1230.692,126.988,-49.661,-178.131,5.607,148.424
C07966=1230.687,127.237,-49.682,-178.128,5.608,148.423
C07967=1230.682,127.486,-49.701,-178.126,5.609,148.423
C07968=1230.677,127.735,-49.722,-178.123,5.610,148.422
C07969=1230.673,127.984,-49.743,-178.121,5.611,148.422
C07970=1230.668,128.234,-49.762,-178.118,5.612,148.421
C07971=1230.663,128.482,-49.782,-178.116,5.613,148.421
C07972=1230.658,128.732,-49.802,-178.113,5.614,148.420
C07973=1230.654,128.981,-49.823,-178.111,5.616,148.420
C07974=1230.649,129.230,-49.843,-178.108,5.616,148.419
C07975=1230.644,129.480,-49.863,-178.105,5.617,148.418
C07976=1230.640,129.728,-49.884,-178.103,5.618,148.418
C07977=1230.635,129.977,-49.904,-178.100,5.620,148.417
C07978=1230.630,130.227,-49.924,-178.098,5.621,148.417
C07979=1230.625,130.476,-49.944,-178.095,5.621,148.416
C07980=1230.620,130.724,-49.965,-178.093,5.623,148.416
C07981=1230.616,130.973,-49.985,-178.090,5.624,148.415
C07982=1230.611,131.223,-50.005,-178.088,5.625,148.415
C07983=1230.606,131.472,-50.026,-178.085,5.626,148.414
C07984=1230.601,131.721,-50.046,-178.083,5.627,148.414
C07985=1230.597,131.971,-50.066,-178.080,5.628,148.413
C07986=1230.592,132.220,-50.086,-178.077,5.630,148.413
C07987=1230.587,132.469,-50.107,-178.075,5.630,148.412
C07988=1230.583,132.718,-50.127,-178.072,5.631,148.412
C07989=1230.578,132.967,-50.148,-178.069,5.633,148.411
C07990=1230.573,133.216,-50.167,-178.067,5.633,148.411
C07991=1230.568,133.485,-50.190,-178.065,5.634,148.410
C07992=1230.562,133.754,-50.211,-178.062,5.636,148.410
C07993=1230.557,134.022,-50.234,-178.059,5.636,148.409
C07994=1230.553,134.291,-50.256,-178.056,5.638,148.409
C07995=1230.548,134.540,-50.277,-178.054,5.639,148.408
C07996=1230.543,134.790,-50.297,-178.051,5.640,148.407
C07997=1230.538,135.038,-50.317,-178.048,5.641,148.407
C07998=1230.533,135.287,-50.338,-178.046,5.642,148.406
C07999=1230.528,135.536,-50.358,-178.043,5.644,148.406
C08000=1230.524,135.785,-50.378,-178.041,5.644,148.405
C08001=1230.519,136.034,-50.399,-178.038,5.645,148.405
C08002=1230.514,136.283,-50.420,-178.035,5.647,148.404
C08003=1230.510,136.532,-50.440,-178.033,5.648,148.404
C08004=1230.505,136.781,-50.461,-178.031,5.648,148.403
C08005=1230.500,137.031,-50.481,-178.028,5.650,148.403
C08006=1230.495,137.280,-50.502,-178.025,5.651,148.402
C08007=1230.490,137.529,-50.522,-178.023,5.652,148.402
C08008=1230.486,137.778,-50.542,-178.020,5.653,148.401
C08009=1230.481,138.027,-50.563,-178.018,5.654,148.401
C08010=1230.476,138.276,-50.584,-178.015,5.655,148.400
C08011=1230.472,138.526,-50.605,-178.013,5.657,148.400
C08012=1230.467,138.775,-50.625,-178.010,5.657,148.399
C08013=1230.463,139.024,-50.646,-178.007,5.659,148.399
C08014=1230.458,139.274,-50.667,-178.005,5.660,148.398
C08015=1230.453,139.522,-50.687,-178.003,5.661,148.398
C08016=1230.448,139.772,-50.708,-178.000,5.662,148.397
C08017=1230.444,140.020,-50.729,-177.997,5.663,148.397
C08018=1230.439,140.269,-50.750,-177.995,5.664,148.396
C08019=1230.434,140.518,-50.770,-177.992,5.666,148.396
C08020=1230.429,140.768,-50.791,-177.990,5.666,148.395
C08021=1230.425,141.016,-50.812,-177.987,5.667,148.395
C08022=1230.420,141.266,-50.833,-177.984,5.669,148.394
C08023=1230.415,141.515,-50.853,-177.982,5.670,148.394
C08024=1230.410,141.764,-50.874,-177.979,5.671,148.393
C08025=1230.406,142.013,-50.894,-177.977,5.672,148.393
C08026=1230.400,142.262,-50.915,-177.975,5.673,148.392
C08027=1230.397,142.511,-50.937,-177.972,5.675,148.392
C08028=1230.392,142.760,-50.958,-177.970,5.676,148.391
C08029=1230.387,143.009,-50.978,-177.967,5.676,148.391
C08030=1230.382,143.259,-50.999,-177.964,5.678,148.390
C08031=1230.378,143.508,-51.020,-177.962,5.679,148.390
C08032=1230.372,143.757,-51.041,-177.959,5.681,148.389
C08033=1230.368,144.006,-51.062,-177.956,5.681,148.389
C08034=1230.363,144.254,-51.083,-177.954,5.682,148.388
C08035=1230.358,144.504,-51.104,-177.951,5.684,148.388
C08036=1230.354,144.753,-51.124,-177.949,5.685,148.387
C08037=1230.349,145.002,-51.146,-177.946,5.686,148.387
C08038=1230.345,145.251,-51.166,-177.944,5.687,148.386
C08039=1230.340,145.500,-51.187,-177.941,5.688,148.386
C08040=1230.335,145.749,-51.208,-177.939,5.690,148.385
C08041=1230.330,145.998,-51.229,-177.936,5.691,148.385
C08042=1230.326,146.248,-51.251,-177.933,5.692,148.384
C08043=1230.321,146.497,-51.272,-177.931,5.693,148.384
C08044=1230.316,146.745,-51.293,-177.929,5.694,148.383
C08045=1230.311,146.995,-51.314,-177.926,5.696,148.383
C08046=1230.307,147.244,-51.334,-177.923,5.696,148.382
C08047=1230.302,147.492,-51.356,-177.921,5.698,148.382
C08048=1230.297,147.742,-51.377,-177.918,5.699,148.381
C08049=1230.293,147.991,-51.397,-177.916,5.700,148.381
C08050=1230.288,148.240,-51.419,-177.913,5.701,148.380
C08051=1230.283,148.489,-51.440,-177.911,5.702,148.380
C08052=1230.279,148.738,-51.460,-177.908,5.704,148.380
C08053=1230.274,148.987,-51.482,-177.905,5.705,148.379
C08054=1230.269,149.237,-51.504,-177.903,5.707,148.379
C08055=1230.264,149.485,-51.525,-177.900,5.707,148.378
C08056=1230.260,149.734,-51.546,-177.898,5.708,148.378
C08057=1230.255,149.983,-51.567,-177.895,5.710,148.377
C08058=1230.250,150.233,-51.589,-177.893,5.711,148.377
C08059=1230.246,150.482,-51.609,-177.890,5.713,148.376
C08060=1230.241,150.730,-51.631,-177.888,5.713,148.376
C08061=1230.236,150.980,-51.652,-177.885,5.715,148.375
C08062=1230.231,151.228,-51.673,-177.882,5.716,148.375
C08063=1230.226,151.478,-51.695,-177.880,5.717,148.374
C08064=1230.222,151.727,-51.716,-177.877,5.718,148.374
C08065=1230.217,151.976,-51.737,-177.875,5.719,148.373
C08066=1230.212,152.224,-51.758,-177.872,5.721,148.373
C08067=1230.208,152.474,-51.780,-177.870,5.722,148.372
C08068=1230.204,152.723,-51.801,-177.867,5.723,148.372
C08069=1230.198,152.972,-51.822,-177.864,5.724,148.371
C08070=1230.194,153.221,-51.844,-177.862,5.725,148.371
C08071=1230.189,153.470,-51.865,-177.859,5.727,148.370
C08072=1230.184,153.719,-51.886,-177.857,5.728,148.370
C08073=1230.179,153.968,-51.908,-177.854,5.729,148.369
C08074=1230.175,154.218,-51.929,-177.852,5.730,148.369
C08075=1230.170,154.466,-51.951,-177.849,5.732,148.368
C08076=1230.166,154.715,-51.972,-177.847,5.733,148.368
C08077=1230.161,154.965,-51.994,-177.844,5.734,148.367
C08078=1230.156,155.213,-52.015,-177.842,5.735,148.367
C08079=1230.151,155.462,-52.037,-177.839,5.737,148.366
C08080=1230.146,155.711,-52.058,-177.837,5.738,148.366
C08081=1230.143,155.960,-52.079,-177.834,5.739,148.365
C08082=1230.138,156.209,-52.101,-177.831,5.740,148.365
C08083=1230.133,156.458,-52.122,-177.829,5.741,148.365
C08084=1230.128,156.708,-52.144,-177.826,5.743,148.364
C08085=1230.123,156.956,-52.166,-177.824,5.744,148.364
C08086=1230.118,157.205,-52.187,-177.821,5.745,148.363
C08087=1230.114,157.455,-52.209,-177.819,5.746,148.363
C08088=1230.109,157.703,-52.230,-177.816,5.748,148.362
C08089=1230.104,157.952,-52.252,-177.813,5.749,148.362
C08090=1230.100,158.202,-52.273,-177.811,5.751,148.361
C08091=1230.095,158.451,-52.295,-177.809,5.752,148.361
C08092=1230.091,158.700,-52.317,-177.806,5.753,148.360
C08093=1230.086,158.948,-52.338,-177.803,5.754,148.360
C08094=1230.081,159.198,-52.359,-177.800,5.756,148.359
C08095=1230.076,159.466,-52.383,-177.798,5.757,148.359
C08096=1230.071,159.736,-52.407,-177.795,5.758,148.358
C08097=1230.066,160.005,-52.429,-177.792,5.760,148.358
C08098=1230.061,160.274,-52.454,-177.790,5.761,148.357
C08099=1230.056,160.523,-52.476,-177.787,5.762,148.357
C08100=1230.051,160.771,-52.497,-177.785,5.763,148.356
C08101=1230.047,161.021,-52.519,-177.782,5.765,148.356
C08102=1230.042,161.270,-52.540,-177.780,5.766,148.356
C08103=1230.038,161.519,-52.562,-177.777,5.767,148.355
C08104=1230.033,161.768,-52.584,-177.775,5.768,148.355
C08105=1230.028,162.017,-52.606,-177.772,5.770,148.354
C08106=1230.024,162.266,-52.628,-177.769,5.771,148.354
C08107=1230.019,162.515,-52.649,-177.767,5.773,148.353
C08108=1230.015,162.764,-52.671,-177.764,5.773,148.353
C08109=1230.010,163.013,-52.693,-177.761,5.775,148.352
C08110=1230.005,163.262,-52.715,-177.759,5.776,148.352
C08111=1230.000,163.511,-52.737,-177.756,5.778,148.351
C08112=1229.995,163.760,-52.759,-177.754,5.779,148.351
C08113=1229.991,164.009,-52.781,-177.751,5.781,148.351
C08114=1229.986,164.258,-52.803,-177.749,5.781,148.350
C08115=1229.982,164.507,-52.825,-177.746,5.783,148.350
C08116=1229.977,164.756,-52.847,-177.744,5.784,148.349
C08117=1229.972,165.005,-52.869,-177.741,5.786,148.349
C08118=1229.968,165.254,-52.890,-177.739,5.787,148.348
C08119=1229.963,165.503,-52.912,-177.736,5.788,148.348
C08120=1229.958,165.752,-52.935,-177.734,5.789,148.347
C08121=1229.953,166.001,-52.957,-177.731,5.791,148.347
C08122=1229.949,166.250,-52.978,-177.729,5.792,148.347
C08123=1229.944,166.499,-53.000,-177.726,5.793,148.346
C08124=1229.939,166.748,-53.022,-177.723,5.795,148.346
C08125=1229.935,166.997,-53.044,-177.721,5.796,148.345
C08126=1229.930,167.246,-53.066,-177.718,5.798,148.345
C08127=1229.925,167.495,-53.088,-177.716,5.799,148.344
C08128=1229.921,167.743,-53.111,-177.713,5.801,148.344
C08129=1229.916,167.993,-53.133,-177.710,5.801,148.343
C08130=1229.912,168.241,-53.155,-177.708,5.803,148.343
C08131=1229.907,168.491,-53.177,-177.706,5.804,148.342
C08132=1229.902,168.740,-53.199,-177.703,5.806,148.342
C08133=1229.897,168.989,-53.221,-177.700,5.807,148.342
C08134=1229.893,169.238,-53.243,-177.698,5.808,148.341
C08135=1229.889,169.486,-53.265,-177.695,5.809,148.341
C08136=1229.883,169.735,-53.288,-177.693,5.811,148.340
C08137=1229.879,169.985,-53.310,-177.690,5.813,148.340
C08138=1229.874,170.234,-53.332,-177.687,5.813,148.339
C08139=1229.870,170.482,-53.354,-177.685,5.815,148.339
C08140=1229.865,170.732,-53.377,-177.683,5.816,148.338
C08141=1229.860,170.980,-53.399,-177.679,5.818,148.338
C08142=1229.856,171.230,-53.421,-177.677,5.819,148.337
C08143=1229.850,171.478,-53.444,-177.675,5.821,148.337
C08144=1229.846,171.727,-53.466,-177.672,5.821,148.336
C08145=1229.842,171.977,-53.488,-177.669,5.823,148.336
C08146=1229.837,172.225,-53.511,-177.667,5.825,148.336
C08147=1229.832,172.474,-53.533,-177.665,5.826,148.335
C08148=1229.828,172.723,-53.554,-177.662,5.827,148.335
C08149=1229.823,172.972,-53.578,-177.659,5.828,148.334
C08150=1229.819,173.221,-53.600,-177.657,5.830,148.334
C08151=1229.814,173.470,-53.621,-177.654,5.831,148.333
C08152=1229.809,173.719,-53.645,-177.652,5.833,148.333
C08153=1229.804,173.968,-53.667,-177.649,5.834,148.333
C08154=1229.800,174.217,-53.689,-177.646,5.835,148.332
C08155=1229.795,174.466,-53.712,-177.644,5.837,148.332
C08156=1229.790,174.715,-53.734,-177.642,5.838,148.331
C08157=1229.786,174.963,-53.756,-177.639,5.840,148.331
C08158=1229.781,175.213,-53.779,-177.636,5.841,148.330
C08159=1229.776,175.462,-53.801,-177.634,5.842,148.330
C08160=1229.772,175.711,-53.824,-177.631,5.844,148.330
C08161=1229.767,175.959,-53.846,-177.629,5.845,148.329
C08162=1229.762,176.208,-53.869,-177.626,5.847,148.329
C08163=1229.758,176.458,-53.891,-177.624,5.848,148.328
C08164=1229.753,176.706,-53.914,-177.621,5.850,148.328
C08165=1229.748,176.955,-53.936,-177.619,5.850,148.327
C08166=1229.744,177.204,-53.959,-177.616,5.852,148.327
C08167=1229.739,177.453,-53.981,-177.613,5.854,148.327
C08168=1229.735,177.702,-54.004,-177.611,5.855,148.326
C08169=1229.730,177.952,-54.027,-177.608,5.857,148.326
C08170=1229.726,178.200,-54.049,-177.606,5.858,148.325
C08171=1229.720,178.449,-54.072,-177.603,5.859,148.325
C08172=1229.716,178.698,-54.094,-177.600,5.861,148.324
C08173=1229.712,178.947,-54.118,-177.598,5.862,148.324
C08174=1229.707,179.196,-54.139,-177.595,5.864,148.324
C08175=1229.702,179.445,-54.163,-177.593,5.865,148.323
C08176=1229.698,179.694,-54.185,-177.590,5.866,148.323
C08177=1229.693,179.943,-54.208,-177.588,5.868,148.322
C08178=1229.688,180.191,-54.231,-177.585,5.869,148.322
C08179=1229.683,180.441,-54.253,-177.583,5.871,148.322
C08180=1229.679,180.689,-54.276,-177.580,5.872,148.321
C08181=1229.674,180.938,-54.299,-177.578,5.873,148.321
C08182=1229.670,181.187,-54.321,-177.575,5.875,148.320
C08183=1229.665,181.436,-54.344,-177.573,5.876,148.320
C08184=1229.661,181.685,-54.368,-177.570,5.878,148.319
C08185=1229.656,181.934,-54.389,-177.567,5.880,148.319
C08186=1229.651,182.183,-54.413,-177.565,5.881,148.319
C08187=1229.647,182.432,-54.436,-177.562,5.883,148.318
C08188=1229.642,182.681,-54.459,-177.559,5.884,148.318
C08189=1229.638,182.930,-54.481,-177.557,5.885,148.317
C08190=1229.633,183.178,-54.504,-177.554,5.887,148.317
C08191=1229.628,183.427,-54.527,-177.552,5.888,148.317
C08192=1229.624,183.676,-54.550,-177.550,5.890,148.316
C08193=1229.619,183.926,-54.573,-177.547,5.891,148.316
C08194=1229.614,184.174,-54.596,-177.544,5.892,148.315
C08195=1229.610,184.423,-54.619,-177.542,5.894,148.315
C08196=1229.605,184.672,-54.642,-177.539,5.896,148.315
C08197=1229.600,184.921,-54.665,-177.537,5.897,148.314
C08198=1229.596,185.170,-54.687,-177.534,5.898,148.314
C08199=1229.591,185.440,-54.712,-177.531,5.900,148.313
C08200=1229.587,185.709,-54.737,-177.528,5.902,148.313
C08201=1229.581,185.978,-54.763,-177.526,5.903,148.312
C08202=1229.576,186.248,-54.788,-177.523,5.905,148.312
C08203=1229.571,186.497,-54.811,-177.520,5.906,148.311
C08204=1229.567,186.746,-54.834,-177.518,5.908,148.311
C08205=1229.562,186.995,-54.856,-177.516,5.909,148.311
C08206=1229.557,187.244,-54.879,-177.513,5.911,148.310
C08207=1229.553,187.493,-54.902,-177.510,5.912,148.310
C08208=1229.548,187.742,-54.925,-177.508,5.913,148.309
C08209=1229.544,187.991,-54.949,-177.505,5.915,148.309
C08210=1229.539,188.240,-54.972,-177.502,5.917,148.309
C08211=1229.535,188.489,-54.995,-177.500,5.918,148.308
C08212=1229.530,188.737,-55.018,-177.497,5.920,148.308
C08213=1229.525,188.986,-55.041,-177.495,5.922,148.307
C08214=1229.520,189.235,-55.065,-177.492,5.923,148.307
C08215=1229.515,189.484,-55.088,-177.490,5.924,148.307
C08216=1229.512,189.733,-55.111,-177.487,5.926,148.306
C08217=1229.507,189.982,-55.134,-177.485,5.927,148.306
C08218=1229.502,190.231,-55.157,-177.482,5.929,148.305
C08219=1229.497,190.480,-55.181,-177.479,5.931,148.305
C08220=1229.493,190.729,-55.204,-177.477,5.932,148.305
C08221=1229.488,190.977,-55.227,-177.475,5.933,148.304
C08222=1229.483,191.226,-55.250,-177.471,5.935,148.304
C08223=1229.479,191.474,-55.274,-177.469,5.936,148.303
C08224=1229.474,191.723,-55.297,-177.467,5.938,148.303
C08225=1229.470,191.972,-55.321,-177.464,5.940,148.303
C08226=1229.465,192.221,-55.344,-177.462,5.941,148.302
C08227=1229.460,192.470,-55.367,-177.459,5.943,148.302
C08228=1229.456,192.719,-55.390,-177.456,5.944,148.301
C08229=1229.452,192.968,-55.414,-177.454,5.946,148.301
C08230=1229.447,193.217,-55.437,-177.452,5.947,148.301
C08231=1229.443,193.466,-55.461,-177.449,5.949,148.300
C08232=1229.438,193.715,-55.484,-177.446,5.951,148.300
C08233=1229.433,193.964,-55.508,-177.444,5.951,148.299
C08234=1229.428,194.213,-55.531,-177.441,5.953,148.299
C08235=1229.424,194.462,-55.554,-177.438,5.955,148.299
C08236=1229.419,194.710,-55.579,-177.436,5.956,148.298
C08237=1229.415,194.959,-55.602,-177.434,5.958,148.298
C08238=1229.410,195.208,-55.625,-177.431,5.960,148.298
C08239=1229.405,195.457,-55.649,-177.428,5.961,148.297
C08240=1229.401,195.706,-55.673,-177.426,5.962,148.297
C08241=1229.397,195.954,-55.695,-177.423,5.964,148.296
C08242=1229.392,196.203,-55.719,-177.421,5.966,148.296
C08243=1229.387,196.452,-55.742,-177.418,5.967,148.296
C08244=1229.383,196.701,-55.766,-177.416,5.969,148.295
C08245=1229.378,196.950,-55.790,-177.413,5.971,148.295
C08246=1229.374,197.199,-55.813,-177.410,5.972,148.294
C08247=1229.369,197.447,-55.837,-177.408,5.973,148.294
C08248=1229.365,197.696,-55.860,-177.405,5.975,148.294
C08249=1229.360,197.945,-55.884,-177.403,5.977,148.293
C08250=1229.355,198.194,-55.908,-177.400,5.979,148.293
C08251=1229.350,198.443,-55.932,-177.398,5.980,148.292
C08252=1229.346,198.692,-55.956,-177.395,5.981,148.292
C08253=1229.341,198.941,-55.979,-177.392,5.983,148.292
C08254=1229.336,199.190,-56.003,-177.390,5.984,148.291
C08255=1229.332,199.438,-56.027,-177.388,5.986,148.291
C08256=1229.327,199.687,-56.050,-177.385,5.988,148.291
C08257=1229.323,199.935,-56.074,-177.382,5.990,148.290
C08258=1229.318,200.184,-56.097,-177.380,5.991,148.290
C08259=1229.314,200.433,-56.121,-177.378,5.993,148.289
C08260=1229.309,200.682,-56.145,-177.374,5.994,148.289
C08261=1229.305,200.930,-56.169,-177.372,5.996,148.289
C08262=1229.300,201.179,-56.192,-177.370,5.997,148.288
C08263=1229.295,201.429,-56.217,-177.367,5.999,148.288
C08264=1229.291,201.678,-56.241,-177.364,6.001,148.288
C08265=1229.286,201.926,-56.265,-177.362,6.003,148.287
C08266=1229.282,202.175,-56.288,-177.360,6.004,148.287
C08267=1229.277,202.424,-56.312,-177.357,6.006,148.286
C08268=1229.272,202.673,-56.336,-177.354,6.007,148.286
C08269=1229.268,202.921,-56.360,-177.351,6.009,148.286
C08270=1229.263,203.170,-56.384,-177.349,6.010,148.285
C08271=1229.258,203.419,-56.408,-177.347,6.012,148.285
C08272=1229.254,203.668,-56.432,-177.344,6.014,148.285
C08273=1229.250,203.917,-56.455,-177.341,6.016,148.284
C08274=1229.245,204.165,-56.480,-177.339,6.017,148.284
C08275=1229.241,204.414,-56.503,-177.337,6.018,148.283
C08276=1229.236,204.663,-56.528,-177.334,6.020,148.283
C08277=1229.231,204.912,-56.552,-177.331,6.022,148.283
C08278=1229.226,205.161,-56.575,-177.328,6.024,148.282
C08279=1229.223,205.410,-56.599,-177.326,6.025,148.282
C08280=1229.218,205.658,-56.624,-177.323,6.027,148.282
C08281=1229.213,205.908,-56.647,-177.321,6.028,148.281
C08282=1229.208,206.156,-56.672,-177.318,6.030,148.281
C08283=1229.204,206.404,-56.696,-177.316,6.031,148.280
C08284=1229.199,206.653,-56.720,-177.314,6.033,148.280
C08285=1229.195,206.903,-56.744,-177.311,6.035,148.280
C08286=1229.190,207.151,-56.768,-177.308,6.037,148.279
C08287=1229.186,207.400,-56.792,-177.305,6.038,148.279
C08288=1229.181,207.648,-56.817,-177.303,6.039,148.279
C08289=1229.176,207.897,-56.840,-177.300,6.041,148.278
C08290=1229.172,208.147,-56.865,-177.298,6.043,148.278
C08291=1229.167,208.395,-56.889,-177.295,6.045,148.278
C08292=1229.163,208.644,-56.913,-177.293,6.047,148.277
C08293=1229.158,208.892,-56.937,-177.290,6.048,148.277
C08294=1229.154,209.142,-56.962,-177.288,6.050,148.276
C08295=1229.149,209.391,-56.986,-177.285,6.052,148.276
C08296=1229.145,209.639,-57.010,-177.283,6.053,148.276
C08297=1229.140,209.888,-57.035,-177.280,6.055,148.275
C08298=1229.135,210.136,-57.059,-177.278,6.056,148.275
C08299=1229.132,210.385,-57.083,-177.275,6.058,148.275
C08300=1229.126,210.634,-57.108,-177.272,6.060,148.274
C08301=1229.122,210.882,-57.132,-177.269,6.062,148.274
C08302=1229.117,211.132,-57.156,-177.267,6.063,148.274
C08303=1229.113,211.402,-57.182,-177.264,6.065,148.273
C08304=1229.108,211.672,-57.209,-177.262,6.067,148.273
C08305=1229.102,211.943,-57.236,-177.259,6.069,148.273
C08306=1229.097,212.213,-57.262,-177.256,6.071,148.272
C08307=1229.093,212.462,-57.286,-177.253,6.072,148.272
C08308=1229.088,212.711,-57.311,-177.251,6.074,148.271
C08309=1229.084,212.960,-57.335,-177.248,6.075,148.271
C08310=1229.079,213.208,-57.360,-177.246,6.077,148.271
C08311=1229.075,213.457,-57.384,-177.243,6.079,148.270
C08312=1229.070,213.706,-57.409,-177.241,6.081,148.270
C08313=1229.065,213.955,-57.433,-177.238,6.083,148.270
C08314=1229.061,214.204,-57.458,-177.235,6.085,148.269
C08315=1229.057,214.452,-57.483,-177.233,6.086,148.269
C08316=1229.051,214.700,-57.507,-177.231,6.087,148.269
C08317=1229.048,214.950,-57.532,-177.228,6.089,148.268
C08318=1229.043,215.198,-57.556,-177.225,6.091,148.268
C08319=1229.038,215.447,-57.580,-177.223,6.093,148.268
C08320=1229.034,215.696,-57.605,-177.220,6.095,148.267
C08321=1229.029,215.945,-57.630,-177.218,6.096,148.267
C08322=1229.024,216.193,-57.654,-177.215,6.098,148.267
C08323=1229.020,216.442,-57.679,-177.213,6.100,148.266
C08324=1229.015,216.691,-57.704,-177.210,6.101,148.266
C08325=1229.011,216.939,-57.728,-177.207,6.103,148.265
C08326=1229.007,217.188,-57.753,-177.204,6.105,148.265
C08327=1229.002,217.437,-57.777,-177.202,6.107,148.265
C08328=1228.998,217.686,-57.802,-177.200,6.108,148.264
C08329=1228.992,217.935,-57.827,-177.197,6.110,148.264
C08330=1228.988,218.183,-57.852,-177.194,6.112,148.264
C08331=1228.984,218.432,-57.877,-177.192,6.113,148.263
C08332=1228.979,218.681,-57.901,-177.189,6.115,148.263
C08333=1228.975,218.930,-57.926,-177.187,6.117,148.263
C08334=1228.970,219.178,-57.951,-177.184,6.119,148.262
C08335=1228.966,219.426,-57.975,-177.182,6.120,148.262
C08336=1228.961,219.676,-58.000,-177.179,6.122,148.262
C08337=1228.956,219.925,-58.025,-177.177,6.124,148.261
C08338=1228.953,220.173,-58.050,-177.174,6.126,148.261
C08339=1228.947,220.422,-58.075,-177.171,6.128,148.261
C08340=1228.942,220.671,-58.099,-177.169,6.129,148.260
C08341=1228.939,220.919,-58.125,-177.166,6.131,148.260
C08342=1228.934,221.168,-58.149,-177.164,6.132,148.260
C08343=1228.929,221.417,-58.174,-177.161,6.134,148.259
C08344=1228.925,221.665,-58.199,-177.159,6.136,148.259
C08345=1228.921,221.914,-58.224,-177.156,6.138,148.259
C08346=1228.916,222.163,-58.250,-177.154,6.140,148.258
C08347=1228.912,222.412,-58.274,-177.151,6.142,148.258
C08348=1228.907,222.660,-58.299,-177.148,6.144,148.258
C08349=1228.903,222.909,-58.324,-177.146,6.145,148.257
C08350=1228.897,223.158,-58.349,-177.144,6.146,148.257
C08351=1228.894,223.406,-58.374,-177.141,6.148,148.257
C08352=1228.889,223.655,-58.399,-177.138,6.150,148.256
C08353=1228.884,223.903,-58.424,-177.136,6.152,148.256
C08354=1228.879,224.153,-58.449,-177.133,6.154,148.256
C08355=1228.875,224.400,-58.474,-177.131,6.156,148.256
C08356=1228.871,224.650,-58.499,-177.128,6.158,148.255
C08357=1228.866,224.898,-58.525,-177.126,6.160,148.255
C08358=1228.861,225.147,-58.550,-177.124,6.161,148.255
C08359=1228.857,225.395,-58.575,-177.121,6.163,148.254
C08360=1228.853,225.645,-58.599,-177.118,6.165,148.254
C08361=1228.849,225.893,-58.625,-177.116,6.166,148.254
C08362=1228.843,226.142,-58.650,-177.113,6.168,148.253
C08363=1228.839,226.391,-58.676,-177.111,6.170,148.253
C08364=1228.834,226.640,-58.700,-177.108,6.172,148.253
C08365=1228.830,226.888,-58.726,-177.105,6.174,148.252
C08366=1228.826,227.136,-58.751,-177.103,6.176,148.252
C08367=1228.821,227.386,-58.776,-177.101,6.177,148.252
C08368=1228.816,227.634,-58.801,-177.098,6.179,148.251
C08369=1228.812,227.883,-58.826,-177.095,6.181,148.251
C08370=1228.807,228.131,-58.852,-177.093,6.182,148.251
C08371=1228.803,228.380,-58.877,-177.090,6.184,148.250
C08372=1228.798,228.630,-58.902,-177.087,6.186,148.250
C08373=1228.794,228.878,-58.928,-177.085,6.188,148.250
C08374=1228.790,229.126,-58.953,-177.082,6.190,148.249
C08375=1228.785,229.375,-58.978,-177.080,6.192,148.249
C08376=1228.781,229.624,-59.003,-177.077,6.194,148.249
C08377=1228.776,229.872,-59.029,-177.075,6.195,148.249
C08378=1228.772,230.121,-59.055,-177.073,6.197,148.248
C08379=1228.767,230.370,-59.080,-177.070,6.199,148.248
C08380=1228.762,230.618,-59.105,-177.068,6.201,148.248
C08381=1228.758,230.867,-59.131,-177.065,6.203,148.247
C08382=1228.753,231.115,-59.156,-177.062,6.204,148.247
C08383=1228.749,231.364,-59.181,-177.060,6.206,148.247
C08384=1228.744,231.613,-59.207,-177.057,6.208,148.246
C08385=1228.740,231.861,-59.232,-177.054,6.210,148.246
C08386=1228.735,232.110,-59.258,-177.052,6.212,148.246
C08387=1228.731,232.359,-59.284,-177.050,6.214,148.246
C08388=1228.726,232.607,-59.309,-177.048,6.215,148.245
C08389=1228.722,232.857,-59.334,-177.045,6.217,148.245
C08390=1228.718,233.105,-59.360,-177.042,6.219,148.245
C08391=1228.713,233.353,-59.385,-177.040,6.221,148.244
C08392=1228.709,233.602,-59.411,-177.037,6.223,148.244
C08393=1228.704,233.850,-59.436,-177.035,6.224,148.244
C08394=1228.700,234.099,-59.462,-177.032,6.226,148.243
C08395=1228.695,234.348,-59.488,-177.029,6.228,148.243
C08396=1228.691,234.597,-59.514,-177.027,6.230,148.243
C08397=1228.686,234.845,-59.539,-177.025,6.232,148.243
C08398=1228.682,235.094,-59.564,-177.022,6.234,148.242
C08399=1228.677,235.343,-59.590,-177.019,6.236,148.242
C08400=1228.672,235.591,-59.616,-177.017,6.238,148.242
C08401=1228.668,235.840,-59.642,-177.014,6.240,148.241
C08402=1228.663,236.089,-59.667,-177.012,6.241,148.241
C08403=1228.659,236.337,-59.693,-177.009,6.243,148.241
C08404=1228.654,236.586,-59.718,-177.007,6.245,148.240
C08405=1228.650,236.835,-59.744,-177.005,6.247,148.240
C08406=1228.645,237.083,-59.770,-177.002,6.249,148.240
C08407=1228.641,237.354,-59.798,-176.999,6.251,148.240
C08408=1228.636,237.626,-59.826,-176.996,6.253,148.239
C08409=1228.630,237.898,-59.855,-176.994,6.255,148.239
C08410=1228.626,238.169,-59.883,-176.991,6.257,148.239
C08411=1228.622,238.418,-59.909,-176.988,6.259,148.238
C08412=1228.617,238.666,-59.935,-176.986,6.261,148.238
C08413=1228.613,238.915,-59.960,-176.983,6.263,148.238
C08414=1228.608,239.163,-59.986,-176.981,6.265,148.238
C08415=1228.603,239.413,-60.012,-176.978,6.266,148.237
C08416=1228.599,239.661,-60.038,-176.976,6.269,148.237
C08417=1228.595,239.909,-60.064,-176.973,6.270,148.237
C08418=1228.590,240.158,-60.090,-176.971,6.272,148.236
C08419=1228.586,240.406,-60.116,-176.968,6.274,148.236
C08420=1228.581,240.655,-60.142,-176.965,6.276,148.236
C08421=1228.576,240.904,-60.167,-176.963,6.278,148.236
C08422=1228.573,241.152,-60.194,-176.960,6.280,148.235
C08423=1228.568,241.401,-60.220,-176.959,6.281,148.235
C08424=1228.563,241.650,-60.246,-176.956,6.283,148.235
C08425=1228.559,241.898,-60.271,-176.953,6.285,148.234
C08426=1228.555,242.146,-60.298,-176.951,6.287,148.234
C08427=1228.550,242.395,-60.324,-176.948,6.289,148.234
C08428=1228.545,242.644,-60.350,-176.946,6.291,148.234
C08429=1228.541,242.893,-60.376,-176.943,6.293,148.233
C08430=1228.536,243.141,-60.402,-176.941,6.295,148.233
C08431=1228.532,243.389,-60.428,-176.938,6.297,148.233
C08432=1228.527,243.638,-60.454,-176.935,6.298,148.232
C08433=1228.523,243.887,-60.481,-176.933,6.300,148.232
C08434=1228.519,244.135,-60.507,-176.931,6.303,148.232
C08435=1228.514,244.384,-60.533,-176.928,6.304,148.232
C08436=1228.509,244.632,-60.559,-176.926,6.306,148.231
C08437=1228.505,244.881,-60.585,-176.923,6.308,148.231
C08438=1228.501,245.130,-60.611,-176.920,6.310,148.231
C08439=1228.496,245.378,-60.638,-176.918,6.312,148.231
C08440=1228.492,245.627,-60.664,-176.916,6.314,148.230
C08441=1228.488,245.875,-60.690,-176.913,6.316,148.230
C08442=1228.483,246.124,-60.716,-176.910,6.318,148.230
C08443=1228.479,246.372,-60.743,-176.908,6.320,148.230
C08444=1228.473,246.621,-60.769,-176.906,6.322,148.229
C08445=1228.469,246.870,-60.795,-176.903,6.324,148.229
C08446=1228.465,247.118,-60.822,-176.900,6.326,148.229
C08447=1228.460,247.367,-60.847,-176.898,6.328,148.228
C08448=1228.456,247.615,-60.874,-176.896,6.330,148.228
C08449=1228.451,247.864,-60.900,-176.893,6.332,148.228
C08450=1228.447,248.112,-60.927,-176.890,6.334,148.228
C08451=1228.443,248.362,-60.953,-176.888,6.335,148.227
C08452=1228.439,248.610,-60.979,-176.885,6.337,148.227
C08453=1228.434,248.858,-61.007,-176.883,6.340,148.227
C08454=1228.430,249.107,-61.032,-176.880,6.341,148.227
C08455=1228.425,249.356,-61.059,-176.878,6.343,148.226
C08456=1228.420,249.604,-61.085,-176.875,6.345,148.226
C08457=1228.416,249.852,-61.112,-176.873,6.347,148.226
C08458=1228.411,250.101,-61.138,-176.870,6.349,148.226
C08459=1228.407,250.349,-61.165,-176.868,6.351,148.225
C08460=1228.403,250.598,-61.191,-176.865,6.353,148.225
C08461=1228.398,250.847,-61.217,-176.863,6.355,148.225
C08462=1228.394,251.095,-61.244,-176.861,6.357,148.225
C08463=1228.389,251.343,-61.271,-176.858,6.359,148.224
C08464=1228.384,251.593,-61.297,-176.855,6.361,148.224
C08465=1228.380,251.841,-61.324,-176.853,6.363,148.224
C08466=1228.376,252.089,-61.351,-176.851,6.365,148.224
C08467=1228.371,252.338,-61.377,-176.848,6.367,148.223
C08468=1228.367,252.587,-61.404,-176.845,6.369,148.223
C08469=1228.363,252.835,-61.430,-176.843,6.371,148.223
C08470=1228.358,253.083,-61.457,-176.841,6.373,148.223
C08471=1228.353,253.332,-61.483,-176.838,6.375,148.222
C08472=1228.349,253.580,-61.510,-176.835,6.377,148.222
C08473=1228.345,253.829,-61.537,-176.833,6.379,148.222
C08474=1228.340,254.077,-61.564,-176.831,6.381,148.222
C08475=1228.336,254.326,-61.590,-176.828,6.383,148.221
C08476=1228.331,254.575,-61.617,-176.825,6.386,148.221
C08477=1228.327,254.823,-61.644,-176.823,6.388,148.221
C08478=1228.323,255.071,-61.670,-176.820,6.389,148.221
C08479=1228.318,255.320,-61.697,-176.818,6.391,148.220
C08480=1228.313,255.568,-61.725,-176.815,6.393,148.220
C08481=1228.309,255.817,-61.750,-176.813,6.395,148.220
C08482=1228.305,256.066,-61.778,-176.810,6.397,148.220
C08483=1228.300,256.315,-61.805,-176.808,6.399,148.220
C08484=1228.296,256.563,-61.831,-176.805,6.401,148.219
C08485=1228.292,256.812,-61.858,-176.803,6.403,148.219
C08486=1228.287,257.060,-61.885,-176.800,6.405,148.219
C08487=1228.283,257.308,-61.912,-176.798,6.407,148.219
C08488=1228.279,257.557,-61.939,-176.796,6.409,148.218
C08489=1228.274,257.805,-61.966,-176.793,6.411,148.218
C08490=1228.269,258.054,-61.993,-176.791,6.413,148.218
C08491=1228.265,258.302,-62.019,-176.788,6.415,148.218
C08492=1228.261,258.550,-62.047,-176.786,6.417,148.217
C08493=1228.256,258.799,-62.074,-176.783,6.419,148.217
C08494=1228.252,259.048,-62.101,-176.781,6.421,148.217
C08495=1228.247,259.297,-62.128,-176.778,6.424,148.217
C08496=1228.243,259.545,-62.155,-176.776,6.426,148.217
C08497=1228.239,259.793,-62.182,-176.773,6.428,148.216
C08498=1228.234,260.042,-62.209,-176.770,6.430,148.216
C08499=1228.229,260.290,-62.236,-176.768,6.432,148.216
C08500=1228.225,260.539,-62.263,-176.766,6.434,148.216
C08501=1228.221,260.787,-62.289,-176.763,6.436,148.215
C08502=1228.217,261.036,-62.317,-176.761,6.438,148.215
C08503=1228.212,261.285,-62.344,-176.758,6.440,148.215
C08504=1228.207,261.533,-62.371,-176.756,6.442,148.215
C08505=1228.203,261.782,-62.398,-176.754,6.444,148.215
C08506=1228.198,262.030,-62.425,-176.751,6.446,148.214
C08507=1228.194,262.278,-62.453,-176.748,6.448,148.214
C08508=1228.190,262.527,-62.480,-176.746,6.451,148.214
C08509=1228.186,262.775,-62.507,-176.743,6.453,148.214
C08510=1228.181,263.024,-62.534,-176.741,6.455,148.214
C08511=1228.176,263.297,-62.564,-176.738,6.457,148.213
C08512=1228.171,263.569,-62.594,-176.735,6.460,148.213
C08513=1228.166,263.841,-62.624,-176.733,6.461,148.213
C08514=1228.161,264.114,-62.653,-176.730,6.463,148.212
C08515=1228.157,264.362,-62.681,-176.728,6.466,148.212
C08516=1228.153,264.612,-62.708,-176.725,6.468,148.212
C08517=1228.148,264.860,-62.735,-176.722,6.470,148.212
C08518=1228.144,265.108,-62.762,-176.720,6.472,148.212
C08519=1228.139,265.356,-62.790,-176.717,6.474,148.211
C08520=1228.135,265.606,-62.818,-176.715,6.477,148.211
C08521=1228.130,265.854,-62.845,-176.713,6.478,148.211
C08522=1228.126,266.102,-62.872,-176.710,6.480,148.211
C08523=1228.121,266.350,-62.899,-176.708,6.483,148.211
C08524=1228.117,266.599,-62.927,-176.705,6.484,148.210
C08525=1228.113,266.848,-62.955,-176.703,6.487,148.210
C08526=1228.108,267.096,-62.982,-176.700,6.489,148.210
C08527=1228.104,267.344,-63.009,-176.698,6.491,148.210
C08528=1228.099,267.592,-63.037,-176.695,6.493,148.210
C08529=1228.095,267.842,-63.064,-176.693,6.495,148.209
C08530=1228.091,268.089,-63.092,-176.691,6.498,148.209
C08531=1228.086,268.338,-63.119,-176.688,6.499,148.209
C08532=1228.082,268.587,-63.146,-176.686,6.502,148.209
C08533=1228.078,268.835,-63.174,-176.683,6.504,148.209
C08534=1228.073,269.084,-63.201,-176.680,6.506,148.208
C08535=1228.069,269.331,-63.229,-176.678,6.508,148.208
C08536=1228.065,269.581,-63.256,-176.675,6.510,148.208
C08537=1228.061,269.828,-63.284,-176.673,6.513,148.208
C08538=1228.055,270.077,-63.312,-176.671,6.514,148.208
C08539=1228.051,270.326,-63.340,-176.669,6.517,148.208
C08540=1228.047,270.574,-63.367,-176.666,6.519,148.207
C08541=1228.042,270.822,-63.395,-176.663,6.520,148.207
C08542=1228.038,271.071,-63.422,-176.661,6.524,148.207
C08543=1228.034,271.319,-63.450,-176.658,6.525,148.207
C08544=1228.029,271.568,-63.477,-176.656,6.528,148.207
C08545=1228.025,271.817,-63.506,-176.653,6.530,148.206
C08546=1228.020,272.065,-63.533,-176.651,6.532,148.206
C08547=1228.016,272.313,-63.561,-176.649,6.534,148.206
C08548=1228.012,272.562,-63.589,-176.647,6.536,148.206
C08549=1228.007,272.810,-63.616,-176.643,6.539,148.206
C08550=1228.003,273.058,-63.644,-176.641,6.541,148.206
C08551=1227.999,273.307,-63.672,-176.639,6.543,148.205
C08552=1227.994,273.555,-63.699,-176.636,6.545,148.205
C08553=1227.990,273.803,-63.727,-176.634,6.547,148.205
C08554=1227.986,274.052,-63.755,-176.631,6.549,148.205
C08555=1227.980,274.301,-63.783,-176.629,6.552,148.205
C08556=1227.977,274.549,-63.811,-176.626,6.554,148.204
C08557=1227.972,274.797,-63.839,-176.624,6.556,148.204
C08558=1227.968,275.045,-63.867,-176.621,6.558,148.204
C08559=1227.963,275.294,-63.895,-176.619,6.560,148.204
C08560=1227.959,275.542,-63.922,-176.617,6.562,148.204
C08561=1227.955,275.791,-63.951,-176.615,6.564,148.204
C08562=1227.951,276.039,-63.978,-176.611,6.567,148.203
C08563=1227.945,276.288,-64.006,-176.609,6.569,148.203
C08564=1227.942,276.536,-64.034,-176.607,6.571,148.203
C08565=1227.937,276.784,-64.062,-176.605,6.573,148.203
C08566=1227.933,277.033,-64.091,-176.602,6.575,148.203
C08567=1227.928,277.281,-64.118,-176.599,6.578,148.203
C08568=1227.924,277.530,-64.146,-176.597,6.580,148.202
C08569=1227.919,277.778,-64.174,-176.595,6.582,148.202
C08570=1227.916,278.027,-64.202,-176.593,6.584,148.202
C08571=1227.911,278.275,-64.230,-176.590,6.586,148.202
C08572=1227.906,278.523,-64.258,-176.588,6.588,148.202
C08573=1227.902,278.771,-64.287,-176.585,6.591,148.201
C08574=1227.898,279.019,-64.314,-176.583,6.593,148.201
C08575=1227.893,279.268,-64.343,-176.580,6.595,148.201
C08576=1227.889,279.516,-64.371,-176.578,6.598,148.201
C08577=1227.885,279.765,-64.398,-176.575,6.599,148.201
C08578=1227.880,280.013,-64.427,-176.573,6.602,148.201
C08579=1227.876,280.262,-64.455,-176.570,6.604,148.200
C08580=1227.871,280.510,-64.483,-176.568,6.607,148.200
C08581=1227.867,280.759,-64.511,-176.566,6.609,148.200
C08582=1227.862,281.007,-64.540,-176.563,6.611,148.200
C08583=1227.859,281.256,-64.568,-176.561,6.613,148.200
C08584=1227.854,281.503,-64.596,-176.558,6.616,148.200
C08585=1227.850,281.752,-64.624,-176.556,6.618,148.200
C08586=1227.845,282.000,-64.652,-176.553,6.620,148.199
C08587=1227.841,282.248,-64.682,-176.551,6.622,148.199
C08588=1227.837,282.496,-64.709,-176.549,6.624,148.199
C08589=1227.832,282.745,-64.738,-176.546,6.627,148.199
C08590=1227.828,282.993,-64.766,-176.544,6.629,148.199
C08591=1227.824,283.242,-64.795,-176.541,6.631,148.199
C08592=1227.820,283.491,-64.823,-176.539,6.633,148.199
C08593=1227.815,283.739,-64.851,-176.536,6.636,148.199
C08594=1227.811,283.987,-64.879,-176.534,6.638,148.198
C08595=1227.806,284.235,-64.908,-176.532,6.640,148.198
C08596=1227.802,284.484,-64.936,-176.529,6.642,148.198
C08597=1227.797,284.732,-64.965,-176.527,6.645,148.198
C08598=1227.794,284.980,-64.993,-176.524,6.648,148.198
C08599=1227.789,285.229,-65.022,-176.522,6.649,148.198
C08600=1227.784,285.477,-65.050,-176.520,6.652,148.197
C08601=1227.780,285.726,-65.078,-176.517,6.654,148.197
C08602=1227.775,285.973,-65.107,-176.515,6.656,148.197
C08603=1227.772,286.222,-65.136,-176.512,6.659,148.197
C08604=1227.767,286.470,-65.164,-176.510,6.661,148.197
C08605=1227.762,286.719,-65.193,-176.508,6.663,148.197
C08606=1227.759,286.967,-65.222,-176.505,6.665,148.197
C08607=1227.754,287.215,-65.250,-176.502,6.668,148.196
C08608=1227.750,287.464,-65.278,-176.500,6.670,148.196
C08609=1227.745,287.713,-65.307,-176.498,6.672,148.196
C08610=1227.741,287.960,-65.336,-176.495,6.674,148.196
C08611=1227.737,288.209,-65.364,-176.493,6.676,148.196
C08612=1227.732,288.457,-65.392,-176.491,6.680,148.196
C08613=1227.728,288.705,-65.422,-176.488,6.681,148.196
C08614=1227.724,288.954,-65.450,-176.486,6.684,148.196
C08615=1227.719,289.228,-65.482,-176.483,6.687,148.196
C08616=1227.714,289.501,-65.514,-176.481,6.689,148.195
C08617=1227.709,289.776,-65.545,-176.478,6.692,148.195
C08618=1227.704,290.050,-65.577,-176.475,6.694,148.195
C08619=1227.700,290.299,-65.606,-176.473,6.697,148.195
C08620=1227.696,290.546,-65.634,-176.471,6.699,148.195
C08621=1227.691,290.795,-65.663,-176.468,6.701,148.195
C08622=1227.687,291.043,-65.692,-176.466,6.703,148.195
C08623=1227.682,291.291,-65.721,-176.463,6.706,148.195
C08624=1227.679,291.539,-65.750,-176.461,6.708,148.194
C08625=1227.674,291.788,-65.778,-176.459,6.710,148.194
C08626=1227.669,292.036,-65.807,-176.457,6.712,148.194
C08627=1227.665,292.285,-65.836,-176.454,6.715,148.194
C08628=1227.661,292.533,-65.865,-176.451,6.717,148.194
C08629=1227.657,292.782,-65.894,-176.449,6.719,148.194
C08630=1227.652,293.029,-65.923,-176.447,6.722,148.194
C08631=1227.648,293.278,-65.952,-176.444,6.725,148.194
C08632=1227.643,293.526,-65.981,-176.442,6.727,148.193
C08633=1227.640,293.774,-66.010,-176.440,6.729,148.193
C08634=1227.635,294.022,-66.038,-176.438,6.731,148.193
C08635=1227.631,294.271,-66.068,-176.435,6.734,148.193
C08636=1227.626,294.520,-66.096,-176.432,6.736,148.193
C08637=1227.622,294.768,-66.126,-176.430,6.738,148.193
C08638=1227.617,295.015,-66.155,-176.428,6.741,148.193
C08639=1227.613,295.264,-66.183,-176.425,6.744,148.193
C08640=1227.609,295.512,-66.213,-176.423,6.745,148.193
C08641=1227.605,295.761,-66.242,-176.421,6.748,148.193
C08642=1227.600,296.009,-66.270,-176.418,6.751,148.193
C08643=1227.596,296.257,-66.300,-176.416,6.753,148.193
C08644=1227.592,296.505,-66.329,-176.414,6.755,148.192
C08645=1227.587,296.754,-66.358,-176.411,6.757,148.192
C08646=1227.583,297.002,-66.387,-176.409,6.760,148.192
C08647=1227.578,297.250,-66.417,-176.407,6.762,148.192
C08648=1227.575,297.498,-66.445,-176.404,6.765,148.192
C08649=1227.570,297.747,-66.474,-176.402,6.768,148.192
C08650=1227.566,297.995,-66.504,-176.399,6.770,148.192
C08651=1227.562,298.243,-66.533,-176.397,6.772,148.192
C08652=1227.557,298.491,-66.562,-176.395,6.774,148.192
C08653=1227.553,298.739,-66.592,-176.392,6.777,148.192
C08654=1227.548,298.988,-66.620,-176.390,6.779,148.192
C08655=1227.544,299.236,-66.650,-176.388,6.781,148.191
C08656=1227.540,299.485,-66.679,-176.386,6.783,148.191
C08657=1227.536,299.733,-66.709,-176.383,6.786,148.191
C08658=1227.531,299.980,-66.738,-176.381,6.789,148.191
C08659=1227.527,300.229,-66.767,-176.379,6.791,148.191
C08660=1227.522,300.478,-66.796,-176.376,6.794,148.191
C08661=1227.518,300.726,-66.825,-176.374,6.796,148.191
C08662=1227.514,300.974,-66.855,-176.371,6.798,148.191
C08663=1227.510,301.222,-66.884,-176.369,6.800,148.191
C08664=1227.506,301.471,-66.914,-176.367,6.803,148.191
C08665=1227.501,301.718,-66.943,-176.364,6.806,148.191
C08666=1227.497,301.967,-66.972,-176.362,6.808,148.191
C08667=1227.493,302.215,-67.002,-176.360,6.811,148.191
C08668=1227.488,302.463,-67.031,-176.358,6.813,148.191
C08669=1227.484,302.712,-67.061,-176.355,6.815,148.190
C08670=1227.479,302.960,-67.091,-176.352,6.818,148.190
C08671=1227.475,303.208,-67.120,-176.350,6.820,148.190
C08672=1227.471,303.456,-67.150,-176.348,6.822,148.190
C08673=1227.467,303.705,-67.179,-176.346,6.825,148.190
C08674=1227.462,303.952,-67.208,-176.343,6.828,148.190
C08675=1227.458,304.201,-67.238,-176.341,6.830,148.190
C08676=1227.454,304.449,-67.267,-176.339,6.832,148.190
C08677=1227.449,304.697,-67.297,-176.336,6.835,148.190
C08678=1227.445,304.946,-67.327,-176.334,6.837,148.190
C08679=1227.441,305.193,-67.357,-176.332,6.840,148.190
C08680=1227.436,305.442,-67.386,-176.330,6.842,148.190
C08681=1227.432,305.690,-67.416,-176.327,6.845,148.190
C08682=1227.428,305.938,-67.445,-176.325,6.847,148.190
C08683=1227.423,306.187,-67.475,-176.323,6.849,148.190
C08684=1227.419,306.435,-67.505,-176.321,6.852,148.190
C08685=1227.415,306.683,-67.534,-176.318,6.854,148.189
C08686=1227.411,306.931,-67.564,-176.316,6.857,148.189
C08687=1227.407,307.179,-67.594,-176.313,6.860,148.189
C08688=1227.402,307.428,-67.624,-176.311,6.862,148.189
C08689=1227.398,307.676,-67.653,-176.309,6.864,148.189
C08690=1227.394,307.924,-67.683,-176.306,6.867,148.189
C08691=1227.390,308.172,-67.713,-176.304,6.869,148.189
C08692=1227.385,308.420,-67.743,-176.302,6.872,148.189
C08693=1227.381,308.669,-67.772,-176.300,6.874,148.189
C08694=1227.376,308.917,-67.802,-176.297,6.877,148.189
C08695=1227.372,309.165,-67.832,-176.295,6.879,148.189
C08696=1227.368,309.413,-67.862,-176.293,6.881,148.189
C08697=1227.363,309.661,-67.891,-176.291,6.884,148.189
C08698=1227.359,309.909,-67.922,-176.288,6.886,148.189
C08699=1227.355,310.158,-67.952,-176.286,6.889,148.189
C08700=1227.350,310.406,-67.981,-176.284,6.892,148.189
C08701=1227.347,310.654,-68.011,-176.282,6.894,148.189
C08702=1227.342,310.902,-68.041,-176.280,6.897,148.189
C08703=1227.337,311.150,-68.071,-176.277,6.900,148.189
C08704=1227.334,311.398,-68.101,-176.275,6.902,148.189
C08705=1227.329,311.647,-68.131,-176.273,6.904,148.189
C08706=1227.325,311.894,-68.161,-176.270,6.907,148.189
C08707=1227.321,312.143,-68.191,-176.268,6.909,148.189
C08708=1227.316,312.391,-68.221,-176.266,6.912,148.189
C08709=1227.312,312.639,-68.251,-176.264,6.915,148.189
C08710=1227.308,312.887,-68.280,-176.261,6.917,148.189
C08711=1227.303,313.135,-68.311,-176.259,6.919,148.189
C08712=1227.299,313.383,-68.341,-176.257,6.922,148.189
C08713=1227.294,313.631,-68.371,-176.255,6.924,148.189
C08714=1227.291,313.880,-68.401,-176.253,6.927,148.189
C08715=1227.287,314.128,-68.431,-176.251,6.929,148.189
C08716=1227.282,314.376,-68.461,-176.248,6.932,148.189
C08717=1227.278,314.624,-68.491,-176.246,6.934,148.189
C08718=1227.273,314.873,-68.522,-176.244,6.937,148.189
C08719=1227.269,315.148,-68.555,-176.241,6.940,148.189
C08720=1227.263,315.424,-68.588,-176.239,6.943,148.189
C08721=1227.259,315.699,-68.622,-176.236,6.946,148.189
C08722=1227.254,315.976,-68.656,-176.234,6.948,148.189
C08723=1227.250,316.223,-68.686,-176.231,6.951,148.189
C08724=1227.246,316.471,-68.717,-176.229,6.953,148.189
C08725=1227.241,316.720,-68.746,-176.228,6.956,148.189
C08726=1227.237,316.968,-68.777,-176.225,6.959,148.189
C08727=1227.234,317.216,-68.807,-176.223,6.961,148.189
C08728=1227.229,317.465,-68.837,-176.221,6.963,148.189
C08729=1227.225,317.712,-68.868,-176.218,6.966,148.189
C08730=1227.220,317.960,-68.898,-176.216,6.969,148.189
C08731=1227.216,318.208,-68.928,-176.214,6.971,148.189
C08732=1227.211,318.456,-68.959,-176.212,6.974,148.189
C08733=1227.207,318.705,-68.990,-176.210,6.976,148.189
C08734=1227.203,318.953,-69.019,-176.207,6.979,148.189
C08735=1227.199,319.201,-69.050,-176.205,6.982,148.189
C08736=1227.195,319.449,-69.080,-176.203,6.984,148.189
C08737=1227.190,319.697,-69.111,-176.201,6.986,148.189
C08738=1227.187,319.946,-69.141,-176.198,6.989,148.189
C08739=1227.182,320.194,-69.171,-176.196,6.992,148.189
C08740=1227.177,320.442,-69.202,-176.195,6.994,148.189
C08741=1227.173,320.689,-69.232,-176.192,6.997,148.189
C08742=1227.169,320.937,-69.263,-176.190,6.999,148.189
C08743=1227.166,321.186,-69.294,-176.188,7.002,148.189
C08744=1227.161,321.434,-69.324,-176.186,7.005,148.189
C08745=1227.156,321.682,-69.354,-176.184,7.007,148.189
C08746=1227.152,321.930,-69.385,-176.181,7.010,148.189
C08747=1227.148,322.179,-69.416,-176.179,7.013,148.189
C08748=1227.143,322.426,-69.447,-176.177,7.015,148.189
C08749=1227.140,322.674,-69.477,-176.175,7.017,148.189
C08750=1227.135,322.922,-69.507,-176.173,7.020,148.189
C08751=1227.131,323.171,-69.539,-176.171,7.023,148.189
C08752=1227.127,323.418,-69.569,-176.169,7.025,148.189
C08753=1227.123,323.666,-69.600,-176.167,7.027,148.189
C08754=1227.118,323.915,-69.630,-176.164,7.031,148.189
C08755=1227.114,324.163,-69.660,-176.162,7.033,148.189
C08756=1227.110,324.411,-69.691,-176.160,7.035,148.189
C08757=1227.105,324.659,-69.722,-176.158,7.039,148.190
C08758=1227.100,324.907,-69.752,-176.156,7.041,148.190
C08759=1227.097,325.156,-69.783,-176.154,7.043,148.189
C08760=1227.093,325.403,-69.814,-176.152,7.046,148.190
C08761=1227.088,325.651,-69.845,-176.150,7.049,148.190
C08762=1227.084,325.899,-69.876,-176.147,7.051,148.190
C08763=1227.080,326.147,-69.906,-176.145,7.054,148.190
C08764=1227.076,326.395,-69.937,-176.143,7.056,148.190
C08765=1227.072,326.644,-69.968,-176.141,7.059,148.190
C08766=1227.067,326.892,-69.999,-176.139,7.062,148.190
C08767=1227.063,327.139,-70.029,-176.137,7.064,148.190
C08768=1227.059,327.388,-70.060,-176.135,7.067,148.190
C08769=1227.055,327.636,-70.091,-176.133,7.070,148.190
C08770=1227.050,327.884,-70.122,-176.130,7.072,148.190
C08771=1227.046,328.133,-70.153,-176.129,7.075,148.190
C08772=1227.042,328.380,-70.185,-176.126,7.078,148.190
C08773=1227.038,328.628,-70.215,-176.125,7.080,148.190
C08774=1227.034,328.876,-70.246,-176.122,7.082,148.190
C08775=1227.029,329.124,-70.277,-176.120,7.086,148.191
C08776=1227.025,329.372,-70.307,-176.118,7.088,148.191
C08777=1227.021,329.620,-70.339,-176.116,7.090,148.191
C08778=1227.016,329.868,-70.370,-176.114,7.094,148.191
C08779=1227.012,330.116,-70.401,-176.112,7.096,148.191
C08780=1227.008,330.364,-70.431,-176.110,7.098,148.191
C08781=1227.004,330.612,-70.463,-176.107,7.101,148.191
C08782=1227.000,330.860,-70.494,-176.106,7.104,148.191
C08783=1226.995,331.108,-70.525,-176.104,7.106,148.191
C08784=1226.991,331.356,-70.555,-176.102,7.109,148.191
C08785=1226.987,331.604,-70.587,-176.099,7.112,148.191
C08786=1226.983,331.852,-70.618,-176.098,7.114,148.191
C08787=1226.978,332.100,-70.649,-176.095,7.117,148.191
C08788=1226.974,332.348,-70.681,-176.094,7.120,148.192
C08789=1226.970,332.596,-70.711,-176.091,7.122,148.192
C08790=1226.966,332.845,-70.743,-176.089,7.125,148.192
C08791=1226.961,333.092,-70.774,-176.087,7.128,148.192
C08792=1226.957,333.341,-70.805,-176.086,7.130,148.192
C08793=1226.953,333.588,-70.837,-176.083,7.134,148.192
C08794=1226.948,333.836,-70.867,-176.081,7.136,148.192
C08795=1226.944,334.085,-70.899,-176.080,7.138,148.192
C08796=1226.940,334.332,-70.930,-176.077,7.141,148.192
C08797=1226.936,334.581,-70.961,-176.075,7.144,148.192
C08798=1226.932,334.828,-70.993,-176.073,7.146,148.192
C08799=1226.928,335.077,-71.024,-176.071,7.149,148.193
C08800=1226.923,335.324,-71.055,-176.069,7.152,148.193
C08801=1226.919,335.573,-71.086,-176.067,7.154,148.193
C08802=1226.915,335.820,-71.118,-176.065,7.158,148.193
C08803=1226.911,336.069,-71.149,-176.063,7.160,148.193
C08804=1226.907,336.316,-71.180,-176.061,7.162,148.193
C08805=1226.903,336.565,-71.212,-176.060,7.165,148.193
C08806=1226.898,336.812,-71.243,-176.057,7.168,148.193
C08807=1226.894,337.060,-71.274,-176.056,7.170,148.194
C08808=1226.890,337.308,-71.306,-176.054,7.173,148.194
C08809=1226.885,337.556,-71.336,-176.051,7.176,148.194
C08810=1226.882,337.804,-71.368,-176.050,7.179,148.194
C08811=1226.876,338.052,-71.400,-176.048,7.181,148.194
C08812=1226.873,338.301,-71.431,-176.045,7.184,148.194
C08813=1226.869,338.549,-71.463,-176.044,7.187,148.194
C08814=1226.864,338.797,-71.494,-176.042,7.189,148.194
C08815=1226.861,339.045,-71.526,-176.039,7.192,148.194
C08816=1226.856,339.292,-71.557,-176.038,7.195,148.195
C08817=1226.852,339.541,-71.589,-176.036,7.197,148.195
C08818=1226.847,339.788,-71.621,-176.034,7.200,148.195
C08819=1226.843,340.037,-71.652,-176.032,7.203,148.195
C08820=1226.839,340.284,-71.683,-176.030,7.205,148.195
C08821=1226.835,340.532,-71.715,-176.029,7.208,148.195
C08822=1226.831,340.780,-71.747,-176.026,7.211,148.195
C08823=1226.826,341.058,-71.781,-176.024,7.214,148.196
C08824=1226.821,341.336,-71.818,-176.022,7.217,148.196
C08825=1226.817,341.614,-71.853,-176.020,7.220,148.196
C08826=1226.812,341.891,-71.888,-176.018,7.223,148.196
C08827=1226.808,342.139,-71.920,-176.016,7.226,148.196
C08828=1226.804,342.387,-71.952,-176.014,7.228,148.196
C08829=1226.799,342.635,-71.983,-176.013,7.231,148.197
C08830=1226.795,342.883,-72.015,-176.010,7.234,148.197
C08831=1226.791,343.130,-72.046,-176.008,7.237,148.197
C08832=1226.787,343.379,-72.079,-176.007,7.239,148.197
C08833=1226.783,343.627,-72.110,-176.005,7.242,148.197
C08834=1226.779,343.874,-72.142,-176.003,7.245,148.197
C08835=1226.775,344.123,-72.173,-176.001,7.247,148.197
C08836=1226.769,344.370,-72.205,-175.999,7.250,148.198
C08837=1226.766,344.618,-72.237,-175.997,7.253,148.198
C08838=1226.762,344.866,-72.269,-175.995,7.256,148.198
C08839=1226.757,345.114,-72.301,-175.994,7.258,148.198
C08840=1226.753,345.362,-72.333,-175.992,7.261,148.198
C08841=1226.749,345.609,-72.364,-175.990,7.264,148.199
C08842=1226.745,345.858,-72.397,-175.988,7.266,148.199
C08843=1226.741,346.106,-72.428,-175.986,7.269,148.199
C08844=1226.736,346.354,-72.459,-175.984,7.272,148.199
C08845=1226.732,346.602,-72.492,-175.982,7.275,148.199
C08846=1226.728,346.850,-72.524,-175.981,7.277,148.199
C08847=1226.724,347.097,-72.555,-175.979,7.280,148.199
C08848=1226.719,347.346,-72.587,-175.977,7.283,148.200
C08849=1226.715,347.593,-72.619,-175.975,7.286,148.200
C08850=1226.711,347.841,-72.651,-175.974,7.288,148.200
C08851=1226.707,348.090,-72.683,-175.972,7.291,148.200
C08852=1226.703,348.337,-72.715,-175.970,7.294,148.200
C08853=1226.698,348.585,-72.747,-175.968,7.297,148.201
C08854=1226.695,348.833,-72.780,-175.967,7.299,148.201
C08855=1226.691,349.081,-72.812,-175.965,7.302,148.201
C08856=1226.686,349.328,-72.844,-175.963,7.305,148.201
C08857=1226.682,349.576,-72.875,-175.961,7.308,148.201
C08858=1226.678,349.825,-72.908,-175.960,7.310,148.202
C08859=1226.674,350.072,-72.939,-175.958,7.313,148.202
C08860=1226.669,350.320,-72.972,-175.956,7.316,148.202
C08861=1226.665,350.568,-73.004,-175.954,7.319,148.202
C08862=1226.660,350.816,-73.036,-175.952,7.321,148.202
C08863=1226.657,351.064,-73.068,-175.951,7.324,148.203
C08864=1226.653,351.312,-73.100,-175.949,7.327,148.203
C08865=1226.649,351.560,-73.133,-175.947,7.329,148.203
C08866=1226.644,351.807,-73.164,-175.945,7.332,148.203
C08867=1226.640,352.056,-73.197,-175.944,7.335,148.203
C08868=1226.636,352.304,-73.228,-175.942,7.338,148.204
C08869=1226.631,352.551,-73.260,-175.940,7.340,148.204
C08870=1226.628,352.799,-73.293,-175.938,7.343,148.204
C08871=1226.623,353.047,-73.325,-175.937,7.345,148.204
C08872=1226.619,353.295,-73.358,-175.935,7.349,148.204
C08873=1226.615,353.543,-73.389,-175.933,7.351,148.205
C08874=1226.611,353.790,-73.422,-175.932,7.354,148.205
C08875=1226.607,354.039,-73.454,-175.930,7.357,148.205
C08876=1226.602,354.287,-73.487,-175.928,7.359,148.205
C08877=1226.598,354.534,-73.518,-175.926,7.363,148.206
C08878=1226.594,354.782,-73.551,-175.925,7.365,148.206
C08879=1226.590,355.030,-73.583,-175.923,7.368,148.206
C08880=1226.586,355.278,-73.616,-175.921,7.370,148.206
C08881=1226.582,355.526,-73.649,-175.920,7.374,148.207
C08882=1226.577,355.773,-73.680,-175.918,7.376,148.207
C08883=1226.573,356.022,-73.713,-175.916,7.379,148.207
C08884=1226.570,356.269,-73.745,-175.915,7.381,148.207
C08885=1226.565,356.518,-73.778,-175.913,7.384,148.207
C08886=1226.561,356.765,-73.811,-175.911,7.388,148.208
C08887=1226.557,357.013,-73.842,-175.910,7.390,148.208
C08888=1226.552,357.261,-73.875,-175.908,7.393,148.208
C08889=1226.549,357.508,-73.907,-175.907,7.395,148.208
C08890=1226.544,357.757,-73.940,-175.905,7.398,148.208
C08891=1226.540,358.004,-73.973,-175.904,7.401,148.209
C08892=1226.536,358.252,-74.004,-175.902,7.404,148.209
C08893=1226.531,358.500,-74.037,-175.900,7.406,148.209
C08894=1226.527,358.748,-74.070,-175.899,7.409,148.210
C08895=1226.524,358.996,-74.102,-175.897,7.412,148.210
C08896=1226.519,359.244,-74.135,-175.896,7.414,148.210
C08897=1226.515,359.492,-74.168,-175.893,7.418,148.210
C08898=1226.512,359.739,-74.200,-175.892,7.421,148.211
C08899=1226.507,359.987,-74.232,-175.891,7.423,148.211
C08900=1226.502,360.235,-74.265,-175.889,7.426,148.211
C08901=1226.499,360.483,-74.297,-175.888,7.428,148.211
C08902=1226.495,360.731,-74.330,-175.886,7.431,148.212
C08903=1226.490,360.979,-74.363,-175.884,7.434,148.212
C08904=1226.486,361.227,-74.396,-175.883,7.437,148.212
C08905=1226.483,361.474,-74.428,-175.881,7.440,148.212
C08906=1226.478,361.722,-74.461,-175.880,7.442,148.213
C08907=1226.473,361.969,-74.494,-175.878,7.445,148.213
C08908=1226.469,362.218,-74.526,-175.877,7.448,148.213
C08909=1226.466,362.465,-74.559,-175.876,7.450,148.214
C08910=1226.461,362.713,-74.592,-175.873,7.454,148.214
C08911=1226.457,362.961,-74.624,-175.872,7.456,148.214
C08912=1226.453,363.209,-74.657,-175.871,7.459,148.214
C08913=1226.449,363.457,-74.689,-175.869,7.462,148.215
C08914=1226.445,363.705,-74.722,-175.868,7.464,148.215
C08915=1226.441,363.952,-74.756,-175.866,7.467,148.215
C08916=1226.436,364.200,-74.788,-175.865,7.470,148.216
C08917=1226.432,364.448,-74.821,-175.863,7.472,148.216
C08918=1226.428,364.695,-74.853,-175.862,7.476,148.216
C08919=1226.424,364.943,-74.887,-175.860,7.478,148.216
C08920=1226.420,365.191,-74.919,-175.859,7.481,148.217
C08921=1226.416,365.439,-74.952,-175.857,7.484,148.217
C08922=1226.411,365.687,-74.985,-175.856,7.487,148.217
C08923=1226.408,365.935,-75.017,-175.854,7.489,148.218
C08924=1226.404,366.183,-75.050,-175.853,7.492,148.218
C08925=1226.399,366.430,-75.083,-175.852,7.495,148.218
C08926=1226.395,366.678,-75.117,-175.850,7.497,148.219
C08927=1226.390,366.958,-75.153,-175.848,7.501,148.219
C08928=1226.386,367.238,-75.191,-175.847,7.504,148.219
C08929=1226.381,367.516,-75.228,-175.845,7.507,148.220
C08930=1226.376,367.797,-75.264,-175.844,7.510,148.220
C08931=1226.372,368.044,-75.298,-175.843,7.513,148.220
C08932=1226.368,368.292,-75.331,-175.841,7.515,148.220
C08933=1226.364,368.540,-75.364,-175.840,7.518,148.221
C08934=1226.360,368.787,-75.397,-175.839,7.521,148.221
C08935=1226.356,369.035,-75.430,-175.837,7.523,148.221
C08936=1226.351,369.284,-75.463,-175.836,7.526,148.222
C08937=1226.347,369.531,-75.496,-175.835,7.529,148.222
C08938=1226.343,369.779,-75.529,-175.833,7.531,148.222
C08939=1226.339,370.027,-75.562,-175.832,7.534,148.223
C08940=1226.335,370.274,-75.595,-175.830,7.537,148.223
C08941=1226.331,370.522,-75.628,-175.829,7.540,148.223
C08942=1226.327,370.770,-75.661,-175.828,7.542,148.224
C08943=1226.323,371.017,-75.694,-175.826,7.545,148.224
C08944=1226.319,371.265,-75.727,-175.825,7.548,148.224
C08945=1226.315,371.513,-75.760,-175.824,7.551,148.225
C08946=1226.311,371.761,-75.794,-175.823,7.553,148.225
C08947=1226.307,372.008,-75.827,-175.821,7.556,148.225
C08948=1226.302,372.256,-75.860,-175.820,7.559,148.226
C08949=1226.298,372.504,-75.893,-175.819,7.562,148.226
C08950=1226.294,372.751,-75.926,-175.818,7.564,148.227
C08951=1226.290,372.999,-75.959,-175.816,7.567,148.227
C08952=1226.286,373.247,-75.992,-175.815,7.570,148.227
C08953=1226.282,373.495,-76.026,-175.814,7.573,148.228
C08954=1226.278,373.743,-76.059,-175.812,7.575,148.228
C08955=1226.274,373.991,-76.092,-175.811,7.578,148.228
C08956=1226.269,374.239,-76.126,-175.810,7.581,148.229
C08957=1226.265,374.487,-76.159,-175.809,7.584,148.229
C08958=1226.261,374.734,-76.192,-175.807,7.586,148.229
C08959=1226.257,374.982,-76.226,-175.806,7.589,148.230
C08960=1226.253,375.230,-76.259,-175.805,7.592,148.230
C08961=1226.248,375.478,-76.292,-175.804,7.594,148.230
C08962=1226.244,375.725,-76.325,-175.803,7.597,148.231
C08963=1226.240,375.973,-76.358,-175.802,7.599,148.231
C08964=1226.236,376.221,-76.391,-175.800,7.602,148.231
C08965=1226.232,376.468,-76.424,-175.799,7.605,148.232
C08966=1226.228,376.716,-76.458,-175.798,7.608,148.232
C08967=1226.224,376.963,-76.491,-175.796,7.610,148.232
C08968=1226.220,377.211,-76.525,-175.795,7.613,148.233
C08969=1226.216,377.459,-76.558,-175.794,7.616,148.233
C08970=1226.211,377.707,-76.592,-175.793,7.618,148.234
C08971=1226.207,377.955,-76.625,-175.792,7.621,148.234
C08972=1226.203,378.202,-76.659,-175.791,7.624,148.234
C08973=1226.199,378.450,-76.692,-175.790,7.627,148.235
C08974=1226.195,378.698,-76.725,-175.789,7.629,148.235
C08975=1226.191,378.945,-76.758,-175.788,7.632,148.236
C08976=1226.187,379.193,-76.792,-175.787,7.634,148.236
C08977=1226.182,379.441,-76.826,-175.785,7.637,148.236
C08978=1226.179,379.689,-76.860,-175.784,7.639,148.237
C08979=1226.175,379.937,-76.893,-175.783,7.642,148.237
C08980=1226.170,380.185,-76.926,-175.782,7.645,148.237
C08981=1226.167,380.432,-76.960,-175.781,7.647,148.238
C08982=1226.163,380.679,-76.993,-175.780,7.650,148.238
C08983=1226.158,380.927,-77.027,-175.779,7.653,148.238
C08984=1226.154,381.175,-77.060,-175.778,7.656,148.239
C08985=1226.150,381.422,-77.094,-175.777,7.658,148.239
C08986=1226.146,381.671,-77.127,-175.776,7.660,148.240
C08987=1226.142,381.918,-77.160,-175.775,7.663,148.240
C08988=1226.137,382.166,-77.195,-175.774,7.666,148.240
C08989=1226.133,382.414,-77.228,-175.772,7.669,148.241
C08990=1226.129,382.661,-77.261,-175.772,7.671,148.241
C08991=1226.125,382.908,-77.295,-175.771,7.674,148.242
C08992=1226.121,383.156,-77.328,-175.769,7.676,148.242
C08993=1226.117,383.405,-77.362,-175.768,7.679,148.242
C08994=1226.113,383.652,-77.396,-175.768,7.681,148.243
C08995=1226.109,383.900,-77.429,-175.766,7.684,148.243
C08996=1226.105,384.147,-77.462,-175.766,7.687,148.244
C08997=1226.100,384.395,-77.497,-175.765,7.690,148.244
C08998=1226.096,384.643,-77.530,-175.764,7.692,148.244
C08999=1226.093,384.890,-77.564,-175.763,7.695,148.245
C09000=1226.088,385.138,-77.598,-175.762,7.698,148.245
C09001=1226.084,385.386,-77.631,-175.761,7.700,148.246
C09002=1226.080,385.633,-77.665,-175.760,7.702,148.246
C09003=1226.076,385.881,-77.698,-175.759,7.705,148.246
C09004=1226.072,386.129,-77.733,-175.758,7.707,148.247
C09005=1226.068,386.377,-77.766,-175.757,7.710,148.247
C09006=1226.064,386.624,-77.800,-175.756,7.713,148.247
C09007=1226.059,386.872,-77.834,-175.755,7.716,148.248
C09008=1226.055,387.120,-77.867,-175.754,7.718,148.248
C09009=1226.052,387.368,-77.901,-175.753,7.721,148.249
C09010=1226.048,387.615,-77.934,-175.752,7.723,148.249
C09011=1226.043,387.863,-77.969,-175.751,7.726,148.250
C09012=1226.039,388.110,-78.002,-175.750,7.728,148.250
C09013=1226.036,388.358,-78.036,-175.749,7.730,148.250
C09014=1226.031,388.606,-78.070,-175.748,7.733,148.251
C09015=1226.027,388.853,-78.104,-175.748,7.736,148.251
C09016=1226.023,389.101,-78.137,-175.747,7.738,148.252
C09017=1226.018,389.349,-78.172,-175.746,7.741,148.252
C09018=1226.015,389.596,-78.206,-175.745,7.743,148.252
C09019=1226.011,389.844,-78.239,-175.744,7.746,148.253
C09020=1226.006,390.091,-78.273,-175.743,7.749,148.253
C09021=1226.002,390.339,-78.307,-175.743,7.751,148.254
C09022=1225.998,390.587,-78.341,-175.741,7.754,148.254
C09023=1225.994,390.835,-78.375,-175.741,7.756,148.254
C09024=1225.990,391.082,-78.408,-175.740,7.759,148.255
C09025=1225.986,391.330,-78.443,-175.738,7.761,148.255
C09026=1225.982,391.578,-78.476,-175.738,7.764,148.256
C09027=1225.978,391.825,-78.511,-175.737,7.767,148.256
C09028=1225.973,392.073,-78.544,-175.736,7.769,148.257
C09029=1225.970,392.320,-78.578,-175.735,7.771,148.257
C09030=1225.966,392.568,-78.613,-175.735,7.773,148.257
C09031=1225.961,392.850,-78.650,-175.734,7.776,148.258
C09032=1225.956,393.131,-78.689,-175.733,7.779,148.258
C09033=1225.951,393.413,-78.728,-175.732,7.782,148.259
C09034=1225.947,393.695,-78.767,-175.731,7.785,148.259
C09035=1225.943,393.942,-78.801,-175.730,7.787,148.260
C09036=1225.938,394.190,-78.835,-175.730,7.790,148.260
C09037=1225.935,394.437,-78.869,-175.729,7.792,148.261
C09038=1225.931,394.685,-78.903,-175.728,7.795,148.261
C09039=1225.926,394.933,-78.936,-175.727,7.797,148.261
C09040=1225.922,395.181,-78.971,-175.726,7.800,148.262
C09041=1225.919,395.428,-79.005,-175.726,7.802,148.262
C09042=1225.914,395.676,-79.038,-175.725,7.805,148.263
C09043=1225.910,395.923,-79.073,-175.724,7.807,148.263
C09044=1225.907,396.171,-79.107,-175.723,7.810,148.264
C09045=1225.902,396.418,-79.141,-175.723,7.812,148.264
C09046=1225.898,396.666,-79.175,-175.721,7.815,148.264
C09047=1225.894,396.914,-79.209,-175.721,7.817,148.265
C09048=1225.890,397.161,-79.243,-175.721,7.819,148.265
C09049=1225.886,397.409,-79.278,-175.719,7.822,148.266
C09050=1225.882,397.657,-79.311,-175.719,7.824,148.266
C09051=1225.877,397.904,-79.346,-175.718,7.827,148.266
C09052=1225.874,398.152,-79.380,-175.717,7.829,148.267
C09053=1225.870,398.400,-79.414,-175.716,7.832,148.267
C09054=1225.866,398.647,-79.448,-175.716,7.834,148.268
C09055=1225.861,398.895,-79.482,-175.715,7.836,148.268
C09056=1225.858,399.143,-79.516,-175.714,7.839,148.269
C09057=1225.853,399.390,-79.551,-175.714,7.841,148.269
C09058=1225.849,399.637,-79.585,-175.713,7.844,148.270
C09059=1225.845,399.885,-79.619,-175.712,7.846,148.270
C09060=1225.841,400.133,-79.654,-175.712,7.848,148.270
C09061=1225.837,400.380,-79.687,-175.710,7.851,148.271
C09062=1225.833,400.629,-79.722,-175.710,7.853,148.271
C09063=1225.829,400.876,-79.756,-175.710,7.855,148.272
C09064=1225.824,401.123,-79.790,-175.708,7.858,148.272
C09065=1225.821,401.371,-79.825,-175.708,7.860,148.272
C09066=1225.816,401.618,-79.859,-175.708,7.862,148.273
C09067=1225.813,401.865,-79.893,-175.706,7.865,148.273
C09068=1225.808,402.114,-79.927,-175.706,7.867,148.274
C09069=1225.804,402.362,-79.961,-175.706,7.869,148.274
C09070=1225.800,402.609,-79.995,-175.705,7.872,148.274
C09071=1225.796,402.857,-80.030,-175.704,7.874,148.275
C09072=1225.792,403.104,-80.064,-175.704,7.876,148.275
C09073=1225.788,403.352,-80.099,-175.703,7.879,148.276
C09074=1225.784,403.599,-80.133,-175.702,7.881,148.276
C09075=1225.780,403.847,-80.167,-175.702,7.883,148.277
C09076=1225.776,404.095,-80.202,-175.701,7.886,148.277
C09077=1225.772,404.342,-80.236,-175.700,7.888,148.278
C09078=1225.767,404.589,-80.270,-175.700,7.890,148.278
C09079=1225.763,404.837,-80.305,-175.699,7.893,148.278
C09080=1225.760,405.084,-80.339,-175.698,7.896,148.279
C09081=1225.756,405.333,-80.374,-175.698,7.898,148.279
C09082=1225.751,405.580,-80.408,-175.697,7.899,148.280
C09083=1225.747,405.827,-80.442,-175.696,7.903,148.280
C09084=1225.743,406.075,-80.477,-175.696,7.905,148.281
C09085=1225.739,406.322,-80.511,-175.695,7.907,148.281
C09086=1225.736,406.570,-80.546,-175.695,7.909,148.281
C09087=1225.731,406.818,-80.580,-175.694,7.912,148.282
C09088=1225.727,407.065,-80.614,-175.693,7.914,148.282
C09089=1225.723,407.313,-80.649,-175.693,7.916,148.283
C09090=1225.719,407.561,-80.683,-175.692,7.918,148.283
C09091=1225.715,407.808,-80.718,-175.691,7.921,148.283
C09092=1225.711,408.056,-80.752,-175.691,7.923,148.284
C09093=1225.706,408.303,-80.787,-175.690,7.925,148.284
C09094=1225.703,408.551,-80.821,-175.690,7.927,148.285
C09095=1225.698,408.798,-80.855,-175.689,7.929,148.285
C09096=1225.694,409.047,-80.890,-175.688,7.932,148.286
C09097=1225.691,409.294,-80.924,-175.688,7.934,148.286
C09098=1225.687,409.542,-80.959,-175.687,7.936,148.286
C09099=1225.682,409.789,-80.993,-175.687,7.938,148.287
C09100=1225.679,410.037,-81.028,-175.686,7.940,148.287
C09101=1225.674,410.284,-81.062,-175.685,7.943,148.288
C09102=1225.670,410.531,-81.097,-175.685,7.945,148.288
C09103=1225.666,410.779,-81.132,-175.684,7.947,148.288
C09104=1225.662,411.026,-81.166,-175.684,7.950,148.289
C09105=1225.658,411.275,-81.201,-175.683,7.952,148.289
C09106=1225.654,411.522,-81.235,-175.683,7.954,148.290
C09107=1225.650,411.770,-81.269,-175.682,7.957,148.290
C09108=1225.646,412.017,-81.304,-175.681,7.959,148.291
C09109=1225.642,412.265,-81.339,-175.681,7.961,148.291
C09110=1225.638,412.512,-81.374,-175.681,7.963,148.291
C09111=1225.634,412.759,-81.408,-175.680,7.965,148.292
C09112=1225.630,413.007,-81.443,-175.679,7.967,148.292
C09113=1225.625,413.255,-81.477,-175.679,7.969,148.293
C09114=1225.621,413.503,-81.512,-175.678,7.972,148.293
C09115=1225.617,413.750,-81.546,-175.677,7.974,148.293
C09116=1225.614,413.998,-81.581,-175.677,7.976,148.294
C09117=1225.609,414.245,-81.616,-175.676,7.978,148.294
C09118=1225.605,414.493,-81.651,-175.676,7.980,148.295
C09119=1225.601,414.740,-81.684,-175.676,7.982,148.295
C09120=1225.597,414.988,-81.719,-175.675,7.984,148.296
C09121=1225.593,415.235,-81.754,-175.674,7.986,148.296
C09122=1225.589,415.483,-81.789,-175.674,7.989,148.296
C09123=1225.583,415.885,-81.846,-175.673,7.993,148.297
C09124=1225.576,416.288,-81.902,-175.672,7.996,148.298
C09125=1225.569,416.690,-81.958,-175.671,8.000,148.298
C09126=1225.565,417.092,-82.014,-175.670,8.003,148.299
